# B&R Automation Studio project A2019059_Linka_Power_CP (part 18)

```iecst
            P1_Robot.KOM_OUT.ManipSrobovania_BezpecnaPozicia:= FALSE;

            P1_Srobovanie.PAR.OsX_ZadanaPozicia:= P1_RemPremenne.P1_Srob5F_PozX_ZadnejSkrutkyM4; //mm
            P1_Srobovanie.PAR.OsY_ZadanaPozicia:= P1_RemPremenne.P1_Srob5F_PozY_ZadnejSkrutkyM4; //mm

            IF NOT SC_P1_Srobovanie.Switch1 AND SC_OvlManipulatora_OsX.Step = 1 AND P1_Srobovacky_VychodziaPozicia AND Safety.STAV.P1_ZonaBunky_AKTIVNA THEN
                OsX_POLOHUJ:= TRUE;
                SC_P1_Srobovanie.Switch1:= TRUE;
            END_IF

            IF NOT SC_P1_Srobovanie.Switch2 AND SC_OvlManipulatora_OsY.Step = 1 AND P1_Srobovacky_VychodziaPozicia AND (P1_Srobovanie.ServoManipulOsX_M20.STATUS.ActualPosition > 14) AND Safety.STAV.P1_ZonaBunky_AKTIVNA THEN
                OsY_POLOHUJ:= TRUE;
                SC_P1_Srobovanie.Switch2:= TRUE;
            END_IF

            IF P1_Srobovanie.STAV.OsX_PoziciaDosiahnuta AND P1_Srobovanie.STAV.OsY_PoziciaDosiahnuta THEN
                P1_Srobovanie.STAV.OsX_PoziciaDosiahnuta:= FALSE;
                P1_Srobovanie.STAV.OsY_PoziciaDosiahnuta:= FALSE;
                IF P1_Srobovanie.RR_PolohujNaPoziciuSkrutky_5F THEN
                    P1_Srobovanie.RR_PolohujNaPoziciuSkrutky_5F:= FALSE;
                    P1_Srobovanie.RR_PolohujNaPoziciuSkrutky_4F:= FALSE;
                    P1_Srobovanie.RR_PolohujNaPoziciuSkrutky_5H:= FALSE;
                    SC_P1_Srobovanie.ResetStep:= TRUE;
                    SC_P1_Srobovanie.Step:= 700;
                ELSE
                    SC_P1_Srobovanie.ResetStep:= TRUE;
                    SC_P1_Srobovanie.Step:= 243;
                END_IF
            END_IF

        243:
            SC_P1_Srobovanie.StepName:='243 - Automaticky Rezim - model 5F, vymazanie vysledkov srobovania';
            SC_P1_Srobovanie.IdleTime.PT:= T#2s;
            SC_P1_Srobovanie.AlarmTime.PT:= T#5s;

            IF NOT SC_P1_Srobovanie.Switch1 THEN
                P1_Srobovanie.Skrutkovacka_M4.RESET_Vysledkov:= TRUE;
                SC_P1_Srobovanie.Switch1:= TRUE;
            END_IF

            IF NOT P1_Srobovanie.Skrutkovacka_M4.Stav_VysledokUtahovania_NG AND NOT P1_Srobovanie.Skrutkovacka_M4.Stav_VysledokUtahovania_OK AND NOT P1_Srobovanie.Skrutkovacka_M4.Stav_UtahovanieUkoncene THEN
                P1_Srobovanie.Skrutkovacka_M4.RESET_Vysledkov:= FALSE;
                SC_P1_Srobovanie.ResetStep:= TRUE;
                SC_P1_Srobovanie.Step:= 245;
            END_IF

        245:
            SC_P1_Srobovanie.StepName:='245 - Automaticky Rezim - model 5F, kontrola skrutky M4 v skrutkovacke';
            SC_P1_Srobovanie.IdleTime.PT:= T#5s;
            SC_P1_Srobovanie.AlarmTime.PT:= T#10s;
            SC_P1_Srobovanie.AlarmTime.IN:= TRUE;

            IF P1_Srobovanie.SkrutkovaciSet_M4.SkrutkaM4_Pripravena AND P1_Srobovanie.Skrutkovacka_M4.Stav_READY_to_START THEN
                SC_P1_Srobovanie.ResetStep:= TRUE;
                SC_P1_Srobovanie.Step:= 248;
            ELSIF SC_P1_Srobovanie.AlarmTime.Q THEN
                IF NOT P1_Srobovanie.Skrutkovacka_M4.Stav_READY_to_START THEN
                    P1_Alarmy[151]:= TRUE;
                    P1_StoperSrobovania.STAV.Porucha:= TRUE;
                    P1_Srobovanie.OUT.KOM_Srobovanie_Ukoncene:= TRUE;
                    SC_P1_Srobovanie.ResetStep:= TRUE;
                    SC_P1_Srobovanie.Step:= 258;
                ELSE
                    FazaNavratu:= 240;
                    SC_P1_Srobovanie.ResetStep:= TRUE;
                    SC_P1_Srobovanie.Step:= 510;
                END_IF
            END_IF

        248:
            SC_P1_Srobovanie.StepName:='248 - Automaticky Rezim - model 5F, vysunutie skrutkovacky M4';
            SC_P1_Srobovanie.IdleTime.PT:= T#500ms;
            SC_P1_Srobovanie.AlarmTime.PT:= T#10s;
            SC_P1_Srobovanie.IdleTime.IN:= TRUE;

            P1_Srobovanie.OUT.SkrutkM4_PrisavSkrutky_RUN_YV81:= TRUE;
            SC_P1_Srobovanie.AlarmTime.IN:= (P1_Srobovanie.IN.SkrutkM4_VysunutieHrotu_IOS10 < 1);

            IF NOT SC_P1_Srobovanie.Switch1 AND SC_P1_Srobovanie.IdleTime.Q THEN
                P1_Srobovanie.OUT.SkrutkM4_VYSUN_YV79:= TRUE;
                P1_Srobovanie.Skrutkovacka_M4.START_Utahovania:= TRUE;
                SC_P1_Srobovanie.Switch1:= TRUE;
            END_IF

            IF NOT P1_Srobovanie.Skrutkovacka_M4.Stav_UtahovanieUkoncene AND P1_Srobovanie.IN.SkrutkM4_VysunutieHrotu_IOS10 > 1 THEN
                SC_P1_Srobovanie.ResetStep:= TRUE;
                SC_P1_Srobovanie.Step:= 250;
            ELSIF SC_P1_Srobovanie.AlarmTime.Q THEN
                P1_Alarmy[144]:= TRUE;
                P1_Srobovanie.OUT.SkrutkM4_VYSUN_YV79:= FALSE;
                P1_Srobovanie.Skrutkovacka_M4.START_Utahovania:= FALSE;
                P1_StoperSrobovania.STAV.Porucha:= TRUE;
                P1_Srobovanie.OUT.KOM_Srobovanie_Ukoncene:= TRUE;
                SC_P1_Srobovanie.ResetStep:= TRUE;
                SC_P1_Srobovanie.Step:= 258;
            END_IF

        250:
            SC_P1_Srobovanie.StepName:='250 - Automaticky Rezim - model 5F, cakam na ukoncenie skrutkovania skrutkovacky M4';
            SC_P1_Srobovanie.IdleTime.PT:= T#30s;
            SC_P1_Srobovanie.AlarmTime.PT:= T#10s;
            SC_P1_Srobovanie.IdleTime.IN:= TRUE;
            SC_P1_Srobovanie.AlarmTime.IN:= TRUE;

            IF P1_Srobovanie.Skrutkovacka_M4.Stav_UtahovanieUkoncene THEN
                P1_Srobovanie.Skrutkovacka_M4.START_Utahovania:= FALSE;
                CasSrobovania:= TIME_TO_REAL(SC_P1_Srobovanie.IdleTime.ET);
                Reports.Skrutkovacky.VyskaSkrutkovania.P1_ZadnaSkrutkaM4:= REAL_TO_STRING(P1_Srobovanie.IN.SkrutkM4_VysunutieHrotu_IOS10);
                Reports.Skrutkovacky.CasSkrutkovania.P1_ZadnaSkrutkaM4:= REAL_TO_STRING(CasSrobovania/1000);
                SC_P1_Srobovanie.ResetStep:= TRUE;
                SC_P1_Srobovanie.Step:= 253;
            ELSIF SC_P1_Srobovanie.AlarmTime.Q THEN
                P1_Alarmy[148]:= TRUE;
                P1_Srobovanie.OUT.SkrutkM4_VYSUN_YV79:= FALSE;
                P1_Srobovanie.Skrutkovacka_M4.START_Utahovania:= FALSE;
                P1_StoperSrobovania.STAV.Porucha:= TRUE;
                P1_Srobovanie.OUT.KOM_Srobovanie_Ukoncene:= TRUE;
                SC_P1_Srobovanie.ResetStep:= TRUE;
                SC_P1_Srobovanie.Step:= 258;
            END_IF

        253:
            SC_P1_Srobovanie.StepName:='253 - Automaticky Rezim - model 5F, zasunutie skrutkovacky M4 a vypnutie prisavania skrutky';
            SC_P1_Srobovanie.IdleTime.PT:= T#200ms;
            SC_P1_Srobovanie.AlarmTime.PT:= T#5s;

            IF NOT SC_P1_Srobovanie.Switch1 THEN
                P1_Srobovanie.OUT.SkrutkM4_VYSUN_YV79:= FALSE;
                P1_Srobovanie.OUT.SkrutkM4_PrisavSkrutky_RUN_YV81:= FALSE;
                SC_P1_Srobovanie.Switch1:= TRUE;
            END_IF

            IF P1_Srobovanie.IN.SkrutkM4_ZASUNUTY_MS17 THEN
                SC_P1_Srobovanie.ResetStep:= TRUE;
                SC_P1_Srobovanie.Step:= 254;
            END_IF

        254:
            SC_P1_Srobovanie.StepName:='254 - Automaticky Rezim - model 5F, signal skrutka M4 odobrata';
            SC_P1_Srobovanie.IdleTime.PT:= T#200ms;
            SC_P1_Srobovanie.AlarmTime.PT:= T#5s;

            IF NOT SC_P1_Srobovanie.Switch1 THEN
                P1_Srobovanie.SkrutkovaciSet_M4.SkrutkaM4_Odobrata:= TRUE;
                SC_P1_Srobovanie.Switch1:= TRUE;
            END_IF

            IF NOT P1_Srobovanie.SkrutkovaciSet_M4.SkrutkaM4_Pripravena THEN
                P1_Srobovanie.SkrutkovaciSet_M4.SkrutkaM4_Odobrata:= FALSE;
                SC_P1_Srobovanie.ResetStep:= TRUE;
                SC_P1_Srobovanie.Step:= 255;
            END_IF

        255:
            SC_P1_Srobovanie.StepName:='255 - Automaticky Rezim - model 5F, kontrola vysledkov skrutkovania zadnej skrutky M4';
            SC_P1_Srobovanie.IdleTime.PT:= T#200ms;
            SC_P1_Srobovanie.AlarmTime.PT:= T#5s;

            IF P1_Srobovanie.Skrutkovacka_M4.Stav_VysledokUtahovania_OK THEN
                P1_Srobovanie.STAV.Vysledok_Srobovania:= 'OK';
                P1_Srobovanie.OUT.KOM_Srobovanie_Ukoncene:= TRUE;
                SC_P1_Srobovanie.ResetStep:= TRUE;
                SC_P1_Srobovanie.Step:= 258;
            ELSIF P1_Srobovanie.Skrutkovacka_M4.Stav_VysledokUtahovania_NG THEN
                P1_Srobovanie.STAV.Vysledok_Srobovania:= 'NG';
                P1_Srobovanie.OUT.KOM_Srobovanie_Ukoncene:= TRUE;
                SC_P1_Srobovanie.ResetStep:= TRUE;
                SC_P1_Srobovanie.Step:= 258;
            END_IF

        258:
            SC_P1_Srobovanie.StepName:='258 - Automaticky Rezim - model 5F, cakam na zrusenie signalu zaskrutkuj zadnu skrutku M4';
            SC_P1_Srobovanie.IdleTime.PT:= T#200ms;
            SC_P1_Srobovanie.AlarmTime.PT:= T#5s;

            IF NOT P1_StoperSrobovania.OUT.KOM_5F_ZasrobujZadnuSkrutku_M4 THEN
                P1_Srobovanie.OUT.KOM_Srobovanie_Ukoncene:= FALSE;
                SC_P1_Srobovanie.ResetStep:= TRUE;
                SC_P1_Srobovanie.Step:= 100;
            END_IF

            //Zaskrutkovanie prednej skrutky M4//

        260:
            SC_P1_Srobovanie.StepName:='260 - Automaticky Rezim - model 5F, napolohovanie zadnej skrutkovacky M4 na poziciu prednej skrutky M4';
            SC_P1_Srobovanie.IdleTime.PT:= T#200ms;
            SC_P1_Srobovanie.AlarmTime.PT:= T#5s;

            P1_Robot.KOM_OUT.ManipSrobovania_BezpecnaPozicia:= FALSE;

            P1_Srobovanie.PAR.OsX_ZadanaPozicia:= P1_RemPremenne.P1_Srob5F_PozX_PrednejSkrutkyM4; //mm
            P1_Srobovanie.PAR.OsY_ZadanaPozicia:= P1_RemPremenne.P1_Srob5F_PozY_PrednejSkrutkyM4; //mm

            IF NOT SC_P1_Srobovanie.Switch1 AND SC_OvlManipulatora_OsX.Step = 1 AND P1_Srobovacky_VychodziaPozicia AND Safety.STAV.P1_ZonaBunky_AKTIVNA THEN
                OsX_POLOHUJ:= TRUE;
                SC_P1_Srobovanie.Switch1:= TRUE;
            END_IF

            IF NOT SC_P1_Srobovanie.Switch2 AND SC_OvlManipulatora_OsY.Step = 1 AND P1_Srobovacky_VychodziaPozicia AND (P1_Srobovanie.ServoManipulOsX_M20.STATUS.ActualPosition > 14) AND Safety.STAV.P1_ZonaBunky_AKTIVNA THEN
                OsY_POLOHUJ:= TRUE;
                SC_P1_Srobovanie.Switch2:= TRUE;
            END_IF

            IF P1_Srobovanie.STAV.OsX_PoziciaDosiahnuta AND P1_Srobovanie.STAV.OsY_PoziciaDosiahnuta THEN
                P1_Srobovanie.STAV.OsX_PoziciaDosiahnuta:= FALSE;
                P1_Srobovanie.STAV.OsY_PoziciaDosiahnuta:= FALSE;
                IF P1_Srobovanie.RR_PolohujNaPoziciuSkrutky_5F THEN
                    P1_Srobovanie.RR_PolohujNaPoziciuSkrutky_5F:= FALSE;
                    P1_Srobovanie.RR_PolohujNaPoziciuSkrutky_4F:= FALSE;
                    P1_Srobovanie.RR_PolohujNaPoziciuSkrutky_5H:= FALSE;
                    SC_P1_Srobovanie.ResetStep:= TRUE;
                    SC_P1_Srobovanie.Step:= 700;
                ELSE
                    SC_P1_Srobovanie.ResetStep:= TRUE;
                    SC_P1_Srobovanie.Step:= 263;
                END_IF
            END_IF

        263:
            SC_P1_Srobovanie.StepName:='263 - Automaticky Rezim - model 5F, vymazanie vysledkov srobovania';
            SC_P1_Srobovanie.IdleTime.PT:= T#2s;
            SC_P1_Srobovanie.AlarmTime.PT:= T#5s;

            IF NOT SC_P1_Srobovanie.Switch1 THEN
                P1_Srobovanie.Skrutkovacka_M4.RESET_Vysledkov:= TRUE;
                SC_P1_Srobovanie.Switch1:= TRUE;
            END_IF

            IF NOT P1_Srobovanie.Skrutkovacka_M4.Stav_VysledokUtahovania_NG AND NOT P1_Srobovanie.Skrutkovacka_M4.Stav_VysledokUtahovania_OK AND NOT P1_Srobovanie.Skrutkovacka_M4.Stav_UtahovanieUkoncene THEN
                P1_Srobovanie.Skrutkovacka_M4.RESET_Vysledkov:= FALSE;
                SC_P1_Srobovanie.ResetStep:= TRUE;
                SC_P1_Srobovanie.Step:= 265;
            END_IF

        265:
            SC_P1_Srobovanie.StepName:='265 - Automaticky Rezim - model 5F, kontrola skrutky M4 v skrutkovacke';
            SC_P1_Srobovanie.IdleTime.PT:= T#5s;
            SC_P1_Srobovanie.AlarmTime.PT:= T#10s;
            SC_P1_Srobovanie.AlarmTime.IN:= TRUE;

            IF P1_Srobovanie.SkrutkovaciSet_M4.SkrutkaM4_Pripravena AND P1_Srobovanie.Skrutkovacka_M4.Stav_READY_to_START THEN
                SC_P1_Srobovanie.ResetStep:= TRUE;
                SC_P1_Srobovanie.Step:= 268;
            ELSIF SC_P1_Srobovanie.AlarmTime.Q THEN
                IF NOT P1_Srobovanie.Skrutkovacka_M4.Stav_READY_to_START THEN
                    P1_Alarmy[151]:= TRUE;
                    P1_StoperSrobovania.STAV.Porucha:= TRUE;
                    P1_Srobovanie.OUT.KOM_Srobovanie_Ukoncene:= TRUE;
                    SC_P1_Srobovanie.ResetStep:= TRUE;
                    SC_P1_Srobovanie.Step:= 278;
                ELSE
                    FazaNavratu:= 260;
                    SC_P1_Srobovanie.ResetStep:= TRUE;
                    SC_P1_Srobovanie.Step:= 510;
                END_IF
            END_IF

        268:
            SC_P1_Srobovanie.StepName:='268 - Automaticky Rezim - model 5F, vysunutie skrutkovacky M4';
            SC_P1_Srobovanie.IdleTime.PT:= T#500ms;
            SC_P1_Srobovanie.AlarmTime.PT:= T#10s;
            SC_P1_Srobovanie.IdleTime.IN:= TRUE;

            P1_Srobovanie.OUT.SkrutkM4_PrisavSkrutky_RUN_YV81:= TRUE;
            SC_P1_Srobovanie.AlarmTime.IN:= (P1_Srobovanie.IN.SkrutkM4_VysunutieHrotu_IOS10 < 1);

            IF NOT SC_P1_Srobovanie.Switch1 AND SC_P1_Srobovanie.IdleTime.Q THEN
                P1_Srobovanie.OUT.SkrutkM4_VYSUN_YV79:= TRUE;
                P1_Srobovanie.Skrutkovacka_M4.START_Utahovania:= TRUE;
                SC_P1_Srobovanie.Switch1:= TRUE;
            END_IF

            IF NOT P1_Srobovanie.Skrutkovacka_M4.Stav_UtahovanieUkoncene AND P1_Srobovanie.IN.SkrutkM4_VysunutieHrotu_IOS10 > 1 THEN
                SC_P1_Srobovanie.ResetStep:= TRUE;
                SC_P1_Srobovanie.Step:= 270;
            ELSIF SC_P1_Srobovanie.AlarmTime.Q THEN
                P1_Alarmy[144]:= TRUE;
                P1_Srobovanie.OUT.SkrutkM4_VYSUN_YV79:= FALSE;
                P1_Srobovanie.Skrutkovacka_M4.START_Utahovania:= FALSE;
                P1_StoperSrobovania.STAV.Porucha:= TRUE;
                P1_Srobovanie.OUT.KOM_Srobovanie_Ukoncene:= TRUE;
                SC_P1_Srobovanie.ResetStep:= TRUE;
                SC_P1_Srobovanie.Step:= 278;
            END_IF

        270:
            SC_P1_Srobovanie.StepName:='270 - Automaticky Rezim - model 5F, cakam na ukoncenie skrutkovania skrutkovacky M4';
            SC_P1_Srobovanie.IdleTime.PT:= T#30s;
            SC_P1_Srobovanie.AlarmTime.PT:= T#10s;
            SC_P1_Srobovanie.IdleTime.IN:= TRUE;
            SC_P1_Srobovanie.AlarmTime.IN:= TRUE;

            IF P1_Srobovanie.Skrutkovacka_M4.Stav_UtahovanieUkoncene THEN
                P1_Srobovanie.Skrutkovacka_M4.START_Utahovania:= FALSE;
                CasSrobovania:= TIME_TO_REAL(SC_P1_Srobovanie.IdleTime.ET);
                Reports.Skrutkovacky.VyskaSkrutkovania.P1_PrednaSkrutkaM4:= REAL_TO_STRING(P1_Srobovanie.IN.SkrutkM4_VysunutieHrotu_IOS10);
                Reports.Skrutkovacky.CasSkrutkovania.P1_PrednaSkrutkaM4:= REAL_TO_STRING(CasSrobovania/1000);
                SC_P1_Srobovanie.ResetStep:= TRUE;
                SC_P1_Srobovanie.Step:= 273;
            ELSIF SC_P1_Srobovanie.AlarmTime.Q THEN
                P1_Alarmy[148]:= TRUE;
                P1_Srobovanie.OUT.SkrutkM4_VYSUN_YV79:= FALSE;
                P1_Srobovanie.Skrutkovacka_M4.START_Utahovania:= FALSE;
                P1_StoperSrobovania.STAV.Porucha:= TRUE;
                P1_Srobovanie.OUT.KOM_Srobovanie_Ukoncene:= TRUE;
                SC_P1_Srobovanie.ResetStep:= TRUE;
                SC_P1_Srobovanie.Step:= 278;
            END_IF

        273:
            SC_P1_Srobovanie.StepName:='273 - Automaticky Rezim - model 5F, zasunutie skrutkovacky M4 a vypnutie prisavania skrutky';
            SC_P1_Srobovanie.IdleTime.PT:= T#200ms;
            SC_P1_Srobovanie.AlarmTime.PT:= T#5s;

            IF NOT SC_P1_Srobovanie.Switch1 THEN
                P1_Srobovanie.OUT.SkrutkM4_VYSUN_YV79:= FALSE;
                P1_Srobovanie.OUT.SkrutkM4_PrisavSkrutky_RUN_YV81:= FALSE;
                SC_P1_Srobovanie.Switch1:= TRUE;
            END_IF

            IF P1_Srobovanie.IN.SkrutkM4_ZASUNUTY_MS17 THEN
                SC_P1_Srobovanie.ResetStep:= TRUE;
                SC_P1_Srobovanie.Step:= 274;
            END_IF

        274:
            SC_P1_Srobovanie.StepName:='274 - Automaticky Rezim - model 5F, signal skrutka M4 odobrata';
            SC_P1_Srobovanie.IdleTime.PT:= T#200ms;
            SC_P1_Srobovanie.AlarmTime.PT:= T#5s;

            IF NOT SC_P1_Srobovanie.Switch1 THEN
                P1_Srobovanie.SkrutkovaciSet_M4.SkrutkaM4_Odobrata:= TRUE;
                SC_P1_Srobovanie.Switch1:= TRUE;
            END_IF

            IF NOT P1_Srobovanie.SkrutkovaciSet_M4.SkrutkaM4_Pripravena THEN
                P1_Srobovanie.SkrutkovaciSet_M4.SkrutkaM4_Odobrata:= FALSE;
                SC_P1_Srobovanie.ResetStep:= TRUE;
                SC_P1_Srobovanie.Step:= 275;
            END_IF

        275:
            SC_P1_Srobovanie.StepName:='275 - Automaticky Rezim - model 5F, kontrola vysledkov skrutkovania prednej skrutky M4';
            SC_P1_Srobovanie.IdleTime.PT:= T#200ms;
            SC_P1_Srobovanie.AlarmTime.PT:= T#5s;

            IF P1_Srobovanie.Skrutkovacka_M4.Stav_VysledokUtahovania_OK THEN
                P1_Srobovanie.STAV.Vysledok_Srobovania:= 'OK';
                P1_Srobovanie.OUT.KOM_Srobovanie_Ukoncene:= TRUE;
                SC_P1_Srobovanie.ResetStep:= TRUE;
                SC_P1_Srobovanie.Step:= 278;
            ELSIF P1_Srobovanie.Skrutkovacka_M4.Stav_VysledokUtahovania_NG THEN
                P1_Srobovanie.STAV.Vysledok_Srobovania:= 'NG';
                P1_Srobovanie.OUT.KOM_Srobovanie_Ukoncene:= TRUE;
                SC_P1_Srobovanie.ResetStep:= TRUE;
                SC_P1_Srobovanie.Step:= 278;
            END_IF

        278:
            SC_P1_Srobovanie.StepName:='278 - Automaticky Rezim - model 5F, cakam na zrusenie signalu zaskrutkuj prednu skrutku M4';
            SC_P1_Srobovanie.IdleTime.PT:= T#200ms;
            SC_P1_Srobovanie.AlarmTime.PT:= T#5s;

            IF NOT P1_StoperSrobovania.OUT.KOM_5F_ZasrobujPrednuSkrutku_M4 THEN
                P1_Srobovanie.OUT.KOM_Srobovanie_Ukoncene:= FALSE;
                SC_P1_Srobovanie.ResetStep:= TRUE;
                SC_P1_Srobovanie.Step:= 100;
            END_IF

            //Zaskrutkovanie skrutky M4 pre DPS//

        280:
            SC_P1_Srobovanie.StepName:='280 - Automaticky Rezim - model 5F, napolohovanie zadnej skrutkovacky M4 na poziciu  skrutky M4 pre DPS';
            SC_P1_Srobovanie.IdleTime.PT:= T#200ms;
            SC_P1_Srobovanie.AlarmTime.PT:= T#5s;

            P1_Robot.KOM_OUT.ManipSrobovania_BezpecnaPozicia:= FALSE;

            P1_Srobovanie.PAR.OsX_ZadanaPozicia:= P1_RemPremenne.P1_Srob5F_PozX_SkrutkyDPS_M4; //mm
            P1_Srobovanie.PAR.OsY_ZadanaPozicia:= P1_RemPremenne.P1_Srob5F_PozY_SkrutkyDPS_M4; //mm

            IF NOT SC_P1_Srobovanie.Switch1 AND SC_OvlManipulatora_OsX.Step = 1 AND P1_Srobovacky_VychodziaPozicia AND Safety.STAV.P1_ZonaBunky_AKTIVNA THEN
                OsX_POLOHUJ:= TRUE;
                SC_P1_Srobovanie.Switch1:= TRUE;
            END_IF

            IF NOT SC_P1_Srobovanie.Switch2 AND SC_OvlManipulatora_OsY.Step = 1 AND P1_Srobovacky_VychodziaPozicia AND (P1_Srobovanie.ServoManipulOsX_M20.STATUS.ActualPosition > 14) AND Safety.STAV.P1_ZonaBunky_AKTIVNA THEN
                OsY_POLOHUJ:= TRUE;
                SC_P1_Srobovanie.Switch2:= TRUE;
            END_IF

            IF P1_Srobovanie.STAV.OsX_PoziciaDosiahnuta AND P1_Srobovanie.STAV.OsY_PoziciaDosiahnuta THEN
                P1_Srobovanie.STAV.OsX_PoziciaDosiahnuta:= FALSE;
                P1_Srobovanie.STAV.OsY_PoziciaDosiahnuta:= FALSE;
                IF P1_Srobovanie.RR_PolohujNaPoziciuSkrutky_5F THEN
                    P1_Srobovanie.RR_PolohujNaPoziciuSkrutky_5F:= FALSE;
                    P1_Srobovanie.RR_PolohujNaPoziciuSkrutky_4F:= FALSE;
                    P1_Srobovanie.RR_PolohujNaPoziciuSkrutky_5H:= FALSE;
                    SC_P1_Srobovanie.ResetStep:= TRUE;
                    SC_P1_Srobovanie.Step:= 700;
                ELSE
                    SC_P1_Srobovanie.ResetStep:= TRUE;
                    SC_P1_Srobovanie.Step:= 282;
                END_IF
            END_IF

        282:
            SC_P1_Srobovanie.StepName:='282 - Automaticky Rezim - model 5F, vymazanie vysledkov srobovania';
            SC_P1_Srobovanie.IdleTime.PT:= T#2s;
            SC_P1_Srobovanie.AlarmTime.PT:= T#5s;

            IF NOT SC_P1_Srobovanie.Switch1 THEN
                P1_Srobovanie.Skrutkovacka_M4.RESET_Vysledkov:= TRUE;
                SC_P1_Srobovanie.Switch1:= TRUE;
            END_IF

            IF NOT P1_Srobovanie.Skrutkovacka_M4.Stav_VysledokUtahovania_NG AND NOT P1_Srobovanie.Skrutkovacka_M4.Stav_VysledokUtahovania_OK AND NOT P1_Srobovanie.Skrutkovacka_M4.Stav_UtahovanieUkoncene THEN
                P1_Srobovanie.Skrutkovacka_M4.RESET_Vysledkov:= FALSE;
                SC_P1_Srobovanie.ResetStep:= TRUE;
                SC_P1_Srobovanie.Step:= 283;
            END_IF

        283:
            SC_P1_Srobovanie.StepName:='283 - Automaticky Rezim - model 5F, kontrola skrutky M4 v skrutkovacke';
            SC_P1_Srobovanie.IdleTime.PT:= T#5s;
            SC_P1_Srobovanie.AlarmTime.PT:= T#10s;
            SC_P1_Srobovanie.AlarmTime.IN:= TRUE;

            IF P1_Srobovanie.SkrutkovaciSet_M4.SkrutkaM4_Pripravena AND P1_Srobovanie.Skrutkovacka_M4.Stav_READY_to_START THEN
                SC_P1_Srobovanie.ResetStep:= TRUE;
                SC_P1_Srobovanie.Step:= 284;
            ELSIF SC_P1_Srobovanie.AlarmTime.Q THEN
                IF NOT P1_Srobovanie.Skrutkovacka_M4.Stav_READY_to_START THEN
                    P1_Alarmy[151]:= TRUE;
                    P1_StoperSrobovania.STAV.Porucha:= TRUE;
                    P1_Srobovanie.OUT.KOM_Srobovanie_Ukoncene:= TRUE;
                    SC_P1_Srobovanie.ResetStep:= TRUE;
                    SC_P1_Srobovanie.Step:= 289;
                ELSE
                    FazaNavratu:= 280;
                    SC_P1_Srobovanie.ResetStep:= TRUE;
                    SC_P1_Srobovanie.Step:= 510;
                END_IF
            END_IF

        284:
            SC_P1_Srobovanie.StepName:='284 - Automaticky Rezim - model 5F, vysunutie skrutkovacky M4';
            SC_P1_Srobovanie.IdleTime.PT:= T#500ms;
            SC_P1_Srobovanie.AlarmTime.PT:= T#10s;
            SC_P1_Srobovanie.IdleTime.IN:= TRUE;

            P1_Srobovanie.OUT.SkrutkM4_PrisavSkrutky_RUN_YV81:= TRUE;
            SC_P1_Srobovanie.AlarmTime.IN:= (P1_Srobovanie.IN.SkrutkM4_VysunutieHrotu_IOS10 < 1);

            IF NOT SC_P1_Srobovanie.Switch1 AND SC_P1_Srobovanie.IdleTime.Q THEN
                P1_Srobovanie.OUT.SkrutkM4_VYSUN_YV79:= TRUE;
                P1_Srobovanie.Skrutkovacka_M4.START_Utahovania:= TRUE;
                SC_P1_Srobovanie.Switch1:= TRUE;
            END_IF

            IF NOT P1_Srobovanie.Skrutkovacka_M4.Stav_UtahovanieUkoncene AND P1_Srobovanie.IN.SkrutkM4_VysunutieHrotu_IOS10 > 1 AND NOT TEST THEN
                SC_P1_Srobovanie.ResetStep:= TRUE;
                SC_P1_Srobovanie.Step:= 285;
            ELSIF SC_P1_Srobovanie.AlarmTime.Q AND NOT TEST THEN
                P1_Alarmy[144]:= TRUE;
                P1_Srobovanie.OUT.SkrutkM4_VYSUN_YV79:= FALSE;
                P1_Srobovanie.Skrutkovacka_M4.START_Utahovania:= FALSE;
                P1_StoperSrobovania.STAV.Porucha:= TRUE;
                P1_Srobovanie.OUT.KOM_Srobovanie_Ukoncene:= TRUE;
                SC_P1_Srobovanie.ResetStep:= TRUE;
                SC_P1_Srobovanie.Step:= 289;
            END_IF

        285:
            SC_P1_Srobovanie.StepName:='285 - Automaticky Rezim - model 5F, cakam na ukoncenie skrutkovania skrutkovacky M4';
            SC_P1_Srobovanie.IdleTime.PT:= T#30s;
            SC_P1_Srobovanie.AlarmTime.PT:= T#10s;
            SC_P1_Srobovanie.IdleTime.IN:= TRUE;
            SC_P1_Srobovanie.AlarmTime.IN:= TRUE;

            IF P1_Srobovanie.Skrutkovacka_M4.Stav_UtahovanieUkoncene THEN
                P1_Srobovanie.Skrutkovacka_M4.START_Utahovania:= FALSE;
                CasSrobovania:= TIME_TO_REAL(SC_P1_Srobovanie.IdleTime.ET);
                Reports.Skrutkovacky.VyskaSkrutkovania.P1_SkrutkaDPS_M4:= REAL_TO_STRING(P1_Srobovanie.IN.SkrutkM4_VysunutieHrotu_IOS10);
                Reports.Skrutkovacky.CasSkrutkovania.P1_SkrutkaDPS_M4:= REAL_TO_STRING(CasSrobovania/1000);
                SC_P1_Srobovanie.ResetStep:= TRUE;
                SC_P1_Srobovanie.Step:= 286;
            ELSIF SC_P1_Srobovanie.AlarmTime.Q THEN
                P1_Alarmy[148]:= TRUE;
                P1_Srobovanie.OUT.SkrutkM4_VYSUN_YV79:= FALSE;
                P1_Srobovanie.Skrutkovacka_M4.START_Utahovania:= FALSE;
                P1_StoperSrobovania.STAV.Porucha:= TRUE;
                P1_Srobovanie.OUT.KOM_Srobovanie_Ukoncene:= TRUE;
                SC_P1_Srobovanie.ResetStep:= TRUE;
                SC_P1_Srobovanie.Step:= 289;
            END_IF

        286:
            SC_P1_Srobovanie.StepName:='286 - Automaticky Rezim - model 5F, zasunutie skrutkovacky M4 a vypnutie prisavania skrutky';
            SC_P1_Srobovanie.IdleTime.PT:= T#200ms;
            SC_P1_Srobovanie.AlarmTime.PT:= T#5s;

            IF NOT SC_P1_Srobovanie.Switch1 THEN
                P1_Srobovanie.OUT.SkrutkM4_VYSUN_YV79:= FALSE;
                P1_Srobovanie.OUT.SkrutkM4_PrisavSkrutky_RUN_YV81:= FALSE;
                SC_P1_Srobovanie.Switch1:= TRUE;
            END_IF

            IF P1_Srobovanie.IN.SkrutkM4_ZASUNUTY_MS17 THEN
                SC_P1_Srobovanie.ResetStep:= TRUE;
                SC_P1_Srobovanie.Step:= 287;
            END_IF

        287:
            SC_P1_Srobovanie.StepName:='287 - Automaticky Rezim - model 5F, signal skrutka M4 odobrata';
            SC_P1_Srobovanie.IdleTime.PT:= T#200ms;
            SC_P1_Srobovanie.AlarmTime.PT:= T#5s;

            IF NOT SC_P1_Srobovanie.Switch1 THEN
                P1_Srobovanie.SkrutkovaciSet_M4.SkrutkaM4_Odobrata:= TRUE;
                SC_P1_Srobovanie.Switch1:= TRUE;
            END_IF

            IF NOT P1_Srobovanie.SkrutkovaciSet_M4.SkrutkaM4_Pripravena THEN
                P1_Srobovanie.SkrutkovaciSet_M4.SkrutkaM4_Odobrata:= FALSE;
                SC_P1_Srobovanie.ResetStep:= TRUE;
                SC_P1_Srobovanie.Step:= 288;
            END_IF

        288:
            SC_P1_Srobovanie.StepName:='288 - Automaticky Rezim - model 5F, kontrola vysledkov skrutkovania skrutky M4 pre DPS';
            SC_P1_Srobovanie.IdleTime.PT:= T#200ms;
            SC_P1_Srobovanie.AlarmTime.PT:= T#5s;

            IF P1_Srobovanie.Skrutkovacka_M4.Stav_VysledokUtahovania_OK THEN
                P1_Srobovanie.STAV.Vysledok_Srobovania:= 'OK';
                P1_Srobovanie.OUT.KOM_Srobovanie_Ukoncene:= TRUE;
                SC_P1_Srobovanie.ResetStep:= TRUE;
                SC_P1_Srobovanie.Step:= 289;
            ELSIF P1_Srobovanie.Skrutkovacka_M4.Stav_VysledokUtahovania_NG THEN
                P1_Srobovanie.STAV.Vysledok_Srobovania:= 'NG';
                P1_Srobovanie.OUT.KOM_Srobovanie_Ukoncene:= TRUE;
                SC_P1_Srobovanie.ResetStep:= TRUE;
                SC_P1_Srobovanie.Step:= 289;
            END_IF

        289:
            SC_P1_Srobovanie.StepName:='289 - Automaticky Rezim - model 5F, cakam na zrusenie signalu zaskrutkuj skrutku M4 pre DPS';
            SC_P1_Srobovanie.IdleTime.PT:= T#200ms;
            SC_P1_Srobovanie.AlarmTime.PT:= T#5s;

            IF NOT P1_StoperSrobovania.OUT.KOM_5F_ZasrobujSkrutkuDPS_M4 THEN
                P1_Srobovanie.OUT.KOM_Srobovanie_Ukoncene:= FALSE;
                SC_P1_Srobovanie.ResetStep:= TRUE;
                SC_P1_Srobovanie.Step:= 100;
            END_IF

            //**********************************************************************Model 5H*******************************************************************************************//
            //Zaskrutkovanie lavej skrutky K30//
        300:
            SC_P1_Srobovanie.StepName:='300 - Automaticky Rezim - model 5H, napolohovanie prednej skrutkovacky K30 na poziciu lavej skrutky K30';
            SC_P1_Srobovanie.IdleTime.PT:= T#200ms;
            SC_P1_Srobovanie.AlarmTime.PT:= T#5s;

            P1_Robot.KOM_OUT.ManipSrobovania_BezpecnaPozicia:= FALSE;

            P1_Srobovanie.PAR.OsX_ZadanaPozicia:= P1_RemPremenne.P1_Srob5H_PozX_LavejSkrutkyK30; //mm
            P1_Srobovanie.PAR.OsY_ZadanaPozicia:= P1_RemPremenne.P1_Srob5H_PozY_LavejSkrutkyK30; //mm

            IF NOT SC_P1_Srobovanie.Switch1 AND SC_OvlManipulatora_OsX.Step = 1 AND P1_Srobovacky_VychodziaPozicia AND Safety.STAV.P1_ZonaBunky_AKTIVNA THEN
                OsX_POLOHUJ:= TRUE;
                SC_P1_Srobovanie.Switch1:= TRUE;
            END_IF

            IF NOT SC_P1_Srobovanie.Switch2 AND SC_OvlManipulatora_OsY.Step = 1 AND P1_Srobovacky_VychodziaPozicia AND (P1_Srobovanie.ServoManipulOsX_M20.STATUS.ActualPosition > 14) AND Safety.STAV.P1_ZonaBunky_AKTIVNA THEN
                OsY_POLOHUJ:= TRUE;
                SC_P1_Srobovanie.Switch2:= TRUE;
            END_IF

            IF P1_Srobovanie.STAV.OsX_PoziciaDosiahnuta AND P1_Srobovanie.STAV.OsY_PoziciaDosiahnuta  THEN
                P1_Srobovanie.STAV.OsX_PoziciaDosiahnuta:= FALSE;
                P1_Srobovanie.STAV.OsY_PoziciaDosiahnuta:= FALSE;
                IF P1_Srobovanie.RR_PolohujNaPoziciuSkrutky_5H THEN
                    P1_Srobovanie.RR_PolohujNaPoziciuSkrutky_5H:= FALSE;
                    P1_Srobovanie.RR_PolohujNaPoziciuSkrutky_4F:= FALSE;
                    P1_Srobovanie.RR_PolohujNaPoziciuSkrutky_5F:= FALSE;
                    SC_P1_Srobovanie.ResetStep:= TRUE;
                    SC_P1_Srobovanie.Step:= 700;
                ELSE
                    SC_P1_Srobovanie.ResetStep:= TRUE;
                    SC_P1_Srobovanie.Step:= 303;
                END_IF
            END_IF

        303:
            SC_P1_Srobovanie.StepName:='303 - Automaticky Rezim - model 5H, vymazanie vysledkov srobovania';
            SC_P1_Srobovanie.IdleTime.PT:= T#2s;
            SC_P1_Srobovanie.AlarmTime.PT:= T#5s;

            IF NOT SC_P1_Srobovanie.Switch1 THEN
                P1_Srobovanie.Skrutkovacka_K30.RESET_Vysledkov:= TRUE;
                SC_P1_Srobovanie.Switch1:= TRUE;
            END_IF

            IF NOT P1_Srobovanie.Skrutkovacka_K30.Stav_VysledokUtahovania_NG AND NOT P1_Srobovanie.Skrutkovacka_K30.Stav_VysledokUtahovania_OK AND NOT P1_Srobovanie.Skrutkovacka_K30.Stav_UtahovanieUkoncene THEN
                P1_Srobovanie.Skrutkovacka_K30.RESET_Vysledkov:= FALSE;
                SC_P1_Srobovanie.ResetStep:= TRUE;
                SC_P1_Srobovanie.Step:= 305;
            END_IF

        305:
            SC_P1_Srobovanie.StepName:='305 - Automaticky Rezim - model 5H, kontrola skrutky K30 v skrutkovacke';
            SC_P1_Srobovanie.IdleTime.PT:= T#5s;
            SC_P1_Srobovanie.AlarmTime.PT:= T#10s;
            SC_P1_Srobovanie.AlarmTime.IN:= TRUE;

            IF P1_Srobovanie.SkrutkovaciSet_K30.SkrutkaK30_Pripravena AND P1_Srobovanie.Skrutkovacka_K30.Stav_READY_to_START THEN
                SC_P1_Srobovanie.ResetStep:= TRUE;
                SC_P1_Srobovanie.Step:= 308;
            ELSIF SC_P1_Srobovanie.AlarmTime.Q THEN
                IF NOT P1_Srobovanie.Skrutkovacka_K30.Stav_READY_to_START THEN
                    P1_Alarmy[149]:= TRUE;
                    P1_StoperSrobovania.STAV.Porucha:= TRUE;
                    P1_Srobovanie.OUT.KOM_Srobovanie_Ukoncene:= TRUE;
                    SC_P1_Srobovanie.ResetStep:= TRUE;
                    SC_P1_Srobovanie.Step:= 318;
                ELSE
                    FazaNavratu:= 300;
                    SC_P1_Srobovanie.ResetStep:= TRUE;
                    SC_P1_Srobovanie.Step:= 500;
                END_IF
            END_IF

        308:
            SC_P1_Srobovanie.StepName:='308 - Automaticky Rezim - model 5H, vysunutie skrutkovacky K30';
            SC_P1_Srobovanie.IdleTime.PT:= T#2s;
            SC_P1_Srobovanie.AlarmTime.PT:= T#5s;

            SC_P1_Srobovanie.AlarmTime.IN:= (P1_Srobovanie.IN.SkrutkK30_VysunutieHrotu_IOS8 < 2);

            IF NOT SC_P1_Srobovanie.Switch1 THEN
                P1_Srobovanie.OUT.SkrutkK30_PrisavSkrutky_RUN_YV90:= TRUE;
                P1_Srobovanie.Skrutkovacka_K30.START_Utahovania:= TRUE;
                P1_Srobovanie.OUT.SkrutkK30_VYSUN_YV89:= TRUE;
                SC_P1_Srobovanie.Switch1:= TRUE;
            ELSIF SC_P1_Srobovanie.AlarmTime.Q THEN
                P1_Alarmy[142]:= TRUE;
                P1_Srobovanie.OUT.SkrutkK30_VYSUN_YV89:= FALSE;
                P1_Srobovanie.Skrutkovacka_K30.START_Utahovania:= FALSE;
                P1_StoperSrobovania.STAV.Porucha:= TRUE;
                P1_Srobovanie.OUT.KOM_Srobovanie_Ukoncene:= TRUE;
                SC_P1_Srobovanie.ResetStep:= TRUE;
                SC_P1_Srobovanie.Step:= 318;
            END_IF

            IF NOT P1_Srobovanie.Skrutkovacka_K30.Stav_UtahovanieUkoncene AND P1_Srobovanie.IN.SkrutkK30_VysunutieHrotu_IOS8 > 2 THEN
                SC_P1_Srobovanie.ResetStep:= TRUE;
                SC_P1_Srobovanie.Step:= 310;
            END_IF

        310:
            SC_P1_Srobovanie.StepName:='310 - Automaticky Rezim - model 5H, cakam na ukoncenie skrutkovania skrutkovacky K30';
            SC_P1_Srobovanie.IdleTime.PT:= T#30s;
            SC_P1_Srobovanie.AlarmTime.PT:= T#10s;
            SC_P1_Srobovanie.IdleTime.IN:= TRUE;
            SC_P1_Srobovanie.AlarmTime.IN:= TRUE;

            IF P1_Srobovanie.Skrutkovacka_K30.Stav_UtahovanieUkoncene THEN
                P1_Srobovanie.Skrutkovacka_K30.START_Utahovania:= FALSE;
                CasSrobovania:= TIME_TO_REAL(SC_P1_Srobovanie.IdleTime.ET);
                Reports.Skrutkovacky.VyskaSkrutkovania.P1_LavaSkrutkaK30:= REAL_TO_STRING(P1_Srobovanie.IN.SkrutkK30_VysunutieHrotu_IOS8);
                Reports.Skrutkovacky.CasSkrutkovania.P1_LavaSkrutkaK30:= REAL_TO_STRING(CasSrobovania/1000);
                SC_P1_Srobovanie.ResetStep:= TRUE;
                SC_P1_Srobovanie.Step:= 313;
            ELSIF SC_P1_Srobovanie.AlarmTime.Q THEN
                P1_Alarmy[146]:= TRUE;
                P1_Srobovanie.OUT.SkrutkK30_VYSUN_YV89:= FALSE;
                P1_Srobovanie.Skrutkovacka_K30.START_Utahovania:= FALSE;
                P1_StoperSrobovania.STAV.Porucha:= TRUE;
                P1_Srobovanie.OUT.KOM_Srobovanie_Ukoncene:= TRUE;
                SC_P1_Srobovanie.ResetStep:= TRUE;
                SC_P1_Srobovanie.Step:= 318;
            END_IF

        313:
            SC_P1_Srobovanie.StepName:='313 - Automaticky Rezim - model 5H, zasunutie skrutkovacky K30 a vypnutie prisavania skrutky';
            SC_P1_Srobovanie.IdleTime.PT:= T#200ms;
            SC_P1_Srobovanie.AlarmTime.PT:= T#5s;

            IF NOT SC_P1_Srobovanie.Switch1 THEN
                P1_Srobovanie.OUT.SkrutkK30_VYSUN_YV89:= FALSE;
                P1_Srobovanie.OUT.SkrutkK30_PrisavSkrutky_RUN_YV90:= FALSE;
                SC_P1_Srobovanie.Switch1:= TRUE;
            END_IF

            IF P1_Srobovanie.IN.SkrutkK30_ZASUNUTY_MS20 THEN
                SC_P1_Srobovanie.ResetStep:= TRUE;
                SC_P1_Srobovanie.Step:= 314;
            END_IF

        314:
            SC_P1_Srobovanie.StepName:='314 - Automaticky Rezim - model 5H, signal skrutka K30 odobrata';
            SC_P1_Srobovanie.IdleTime.PT:= T#200ms;
            SC_P1_Srobovanie.AlarmTime.PT:= T#5s;

            IF NOT SC_P1_Srobovanie.Switch1 THEN
                P1_Srobovanie.SkrutkovaciSet_K30.SkrutkaK30_Odobrata:= TRUE;
                SC_P1_Srobovanie.Switch1:= TRUE;
            END_IF

            IF NOT P1_Srobovanie.SkrutkovaciSet_K30.SkrutkaK30_Pripravena THEN
                P1_Srobovanie.SkrutkovaciSet_K30.SkrutkaK30_Odobrata:= FALSE;
                SC_P1_Srobovanie.ResetStep:= TRUE;
                SC_P1_Srobovanie.Step:= 315;
            END_IF

        315:
            SC_P1_Srobovanie.StepName:='315 - Automaticky Rezim - model 5H, kontrola vysledkov skrutkovania lavej skrutky K30';
            SC_P1_Srobovanie.IdleTime.PT:= T#200ms;
            SC_P1_Srobovanie.AlarmTime.PT:= T#5s;

            IF P1_Srobovanie.Skrutkovacka_K30.Stav_VysledokUtahovania_OK THEN
                P1_Srobovanie.STAV.Vysledok_Srobovania:= 'OK';
                P1_Srobovanie.OUT.KOM_Srobovanie_Ukoncene:= TRUE;
                SC_P1_Srobovanie.ResetStep:= TRUE;
                SC_P1_Srobovanie.Step:= 318;
            ELSIF P1_Srobovanie.Skrutkovacka_K30.Stav_VysledokUtahovania_NG THEN
                P1_Srobovanie.STAV.Vysledok_Srobovania:= 'NG';
                P1_Srobovanie.OUT.KOM_Srobovanie_Ukoncene:= TRUE;
                SC_P1_Srobovanie.ResetStep:= TRUE;
                SC_P1_Srobovanie.Step:= 318;
            END_IF

        318:
            SC_P1_Srobovanie.StepName:='318 - Automaticky Rezim - model 5H, cakam na zrusenie signalu zaskrutkuj lavu skrutku K30';
            SC_P1_Srobovanie.IdleTime.PT:= T#200ms;
            SC_P1_Srobovanie.AlarmTime.PT:= T#5s;

            IF NOT P1_StoperSrobovania.OUT.KOM_5H_ZasrobujLavuSkrutku_K30 THEN
                P1_Srobovanie.OUT.KOM_Srobovanie_Ukoncene:= FALSE;
                SC_P1_Srobovanie.ResetStep:= TRUE;
                SC_P1_Srobovanie.Step:= 100;
            END_IF

            //Zaskrutkovanie pravej skrutky K30//

        320:
            SC_P1_Srobovanie.StepName:='320 - Automaticky Rezim - model 5H, napolohovanie prednej skrutkovacky K30 na poziciu pravej skrutky K30';
            SC_P1_Srobovanie.IdleTime.PT:= T#200ms;
            SC_P1_Srobovanie.AlarmTime.PT:= T#5s;

            P1_Robot.KOM_OUT.ManipSrobovania_BezpecnaPozicia:= FALSE;

            P1_Srobovanie.PAR.OsX_ZadanaPozicia:= P1_RemPremenne.P1_Srob5F_PozX_PravejSkrutkyK30; //mm
            P1_Srobovanie.PAR.OsY_ZadanaPozicia:= P1_RemPremenne.P1_Srob5F_PozY_PravejSkrutkyK30; //mm

            IF NOT SC_P1_Srobovanie.Switch1 AND SC_OvlManipulatora_OsX.Step = 1 AND P1_Srobovacky_VychodziaPozicia AND Safety.STAV.P1_ZonaBunky_AKTIVNA THEN
                OsX_POLOHUJ:= TRUE;
                SC_P1_Srobovanie.Switch1:= TRUE;
            END_IF

            IF NOT SC_P1_Srobovanie.Switch2 AND SC_OvlManipulatora_OsY.Step = 1 AND P1_Srobovacky_VychodziaPozicia AND (P1_Srobovanie.ServoManipulOsX_M20.STATUS.ActualPosition > 14) AND Safety.STAV.P1_ZonaBunky_AKTIVNA THEN
                OsY_POLOHUJ:= TRUE;
                SC_P1_Srobovanie.Switch2:= TRUE;
            END_IF

            IF P1_Srobovanie.STAV.OsX_PoziciaDosiahnuta AND P1_Srobovanie.STAV.OsY_PoziciaDosiahnuta  THEN
                P1_Srobovanie.STAV.OsX_PoziciaDosiahnuta:= FALSE;
                P1_Srobovanie.STAV.OsY_PoziciaDosiahnuta:= FALSE;
                IF P1_Srobovanie.RR_PolohujNaPoziciuSkrutky_5H THEN
                    P1_Srobovanie.RR_PolohujNaPoziciuSkrutky_5H:= FALSE;
                    P1_Srobovanie.RR_PolohujNaPoziciuSkrutky_4F:= FALSE;
                    P1_Srobovanie.RR_PolohujNaPoziciuSkrutky_5F:= FALSE;
                    SC_P1_Srobovanie.ResetStep:= TRUE;
                    SC_P1_Srobovanie.Step:= 700;
                ELSE
                    SC_P1_Srobovanie.ResetStep:= TRUE;
                    SC_P1_Srobovanie.Step:= 323;
                END_IF
            END_IF

        323:
            SC_P1_Srobovanie.StepName:='323 - Automaticky Rezim - model 5H, vymazanie vysledkov srobovania';
            SC_P1_Srobovanie.IdleTime.PT:= T#2s;
            SC_P1_Srobovanie.AlarmTime.PT:= T#5s;

            IF NOT SC_P1_Srobovanie.Switch1 THEN
                P1_Srobovanie.Skrutkovacka_K30.RESET_Vysledkov:= TRUE;
                SC_P1_Srobovanie.Switch1:= TRUE;
            END_IF

            IF NOT P1_Srobovanie.Skrutkovacka_K30.Stav_VysledokUtahovania_NG AND NOT P1_Srobovanie.Skrutkovacka_K30.Stav_VysledokUtahovania_OK AND NOT P1_Srobovanie.Skrutkovacka_K30.Stav_UtahovanieUkoncene THEN
                P1_Srobovanie.Skrutkovacka_K30.RESET_Vysledkov:= FALSE;
                SC_P1_Srobovanie.ResetStep:= TRUE;
                SC_P1_Srobovanie.Step:= 325;
            END_IF

        325:
            SC_P1_Srobovanie.StepName:='325 - Automaticky Rezim - model 5H, kontrola skrutky K30 v skrutkovacke';
            SC_P1_Srobovanie.IdleTime.PT:= T#5s;
            SC_P1_Srobovanie.AlarmTime.PT:= T#10s;
            SC_P1_Srobovanie.AlarmTime.IN:= TRUE;

            IF P1_Srobovanie.SkrutkovaciSet_K30.SkrutkaK30_Pripravena AND P1_Srobovanie.Skrutkovacka_K30.Stav_READY_to_START THEN
                SC_P1_Srobovanie.ResetStep:= TRUE;
                SC_P1_Srobovanie.Step:= 328;
            ELSIF SC_P1_Srobovanie.AlarmTime.Q THEN
                IF NOT P1_Srobovanie.Skrutkovacka_K30.Stav_READY_to_START THEN
                    P1_Alarmy[149]:= TRUE;
                    P1_StoperSrobovania.STAV.Porucha:= TRUE;
                    P1_Srobovanie.OUT.KOM_Srobovanie_Ukoncene:= TRUE;
                    SC_P1_Srobovanie.ResetStep:= TRUE;
                    SC_P1_Srobovanie.Step:= 338;
                ELSE
                    FazaNavratu:= 320;
                    SC_P1_Srobovanie.ResetStep:= TRUE;
                    SC_P1_Srobovanie.Step:= 500;
                END_IF
            END_IF

        328:
            SC_P1_Srobovanie.StepName:='328 - Automaticky Rezim - model 5H, vysunutie skrutkovacky K30';
            SC_P1_Srobovanie.IdleTime.PT:= T#2s;
            SC_P1_Srobovanie.AlarmTime.PT:= T#5s;

            SC_P1_Srobovanie.AlarmTime.IN:= (P1_Srobovanie.IN.SkrutkK30_VysunutieHrotu_IOS8 < 2);

            IF NOT SC_P1_Srobovanie.Switch1 THEN
                P1_Srobovanie.OUT.SkrutkK30_PrisavSkrutky_RUN_YV90:= TRUE;
                P1_Srobovanie.Skrutkovacka_K30.START_Utahovania:= TRUE;
                P1_Srobovanie.OUT.SkrutkK30_VYSUN_YV89:= TRUE;
                SC_P1_Srobovanie.Switch1:= TRUE;
            END_IF

            IF NOT P1_Srobovanie.Skrutkovacka_K30.Stav_UtahovanieUkoncene AND P1_Srobovanie.IN.SkrutkK30_VysunutieHrotu_IOS8 > 2 THEN
                SC_P1_Srobovanie.ResetStep:= TRUE;
                SC_P1_Srobovanie.Step:= 330;
            ELSIF SC_P1_Srobovanie.AlarmTime.Q THEN
                P1_Alarmy[142]:= TRUE;
                P1_Srobovanie.OUT.SkrutkK30_VYSUN_YV89:= FALSE;
                P1_Srobovanie.Skrutkovacka_K30.START_Utahovania:= FALSE;
                P1_StoperSrobovania.STAV.Porucha:= TRUE;
                P1_Srobovanie.OUT.KOM_Srobovanie_Ukoncene:= TRUE;
                SC_P1_Srobovanie.ResetStep:= TRUE;
                SC_P1_Srobovanie.Step:= 338;
            END_IF

        330:
            SC_P1_Srobovanie.StepName:='330 - Automaticky Rezim - model 5H, cakam na ukoncenie skrutkovania skrutkovacky K30';
            SC_P1_Srobovanie.IdleTime.PT:= T#30s;
            SC_P1_Srobovanie.AlarmTime.PT:= T#10s;
            SC_P1_Srobovanie.IdleTime.IN:= TRUE;
            SC_P1_Srobovanie.AlarmTime.IN:= TRUE;

            IF P1_Srobovanie.Skrutkovacka_K30.Stav_UtahovanieUkoncene THEN
                P1_Srobovanie.Skrutkovacka_K30.START_Utahovania:= FALSE;
                CasSrobovania:= TIME_TO_REAL(SC_P1_Srobovanie.IdleTime.ET);
                Reports.Skrutkovacky.VyskaSkrutkovania.P1_PravaSkrutkaK30:= REAL_TO_STRING(P1_Srobovanie.IN.SkrutkK30_VysunutieHrotu_IOS8);
                Reports.Skrutkovacky.CasSkrutkovania.P1_PravaSkrutkaK30:= REAL_TO_STRING(CasSrobovania/1000);
                SC_P1_Srobovanie.ResetStep:= TRUE;
                SC_P1_Srobovanie.Step:= 331;
            ELSIF SC_P1_Srobovanie.AlarmTime.Q THEN
                P1_Alarmy[146]:= TRUE;
                P1_Srobovanie.OUT.SkrutkK30_VYSUN_YV89:= FALSE;
                P1_Srobovanie.Skrutkovacka_K30.START_Utahovania:= FALSE;
                P1_StoperSrobovania.STAV.Porucha:= TRUE;
                P1_Srobovanie.OUT.KOM_Srobovanie_Ukoncene:= TRUE;
                SC_P1_Srobovanie.ResetStep:= TRUE;
                SC_P1_Srobovanie.Step:= 338;
            END_IF

        331:
            SC_P1_Srobovanie.StepName:='331 - Automaticky Rezim - model 5H, zasunutie skrutkovacky K30 a vypnutie prisavania skrutky';
            SC_P1_Srobovanie.IdleTime.PT:= T#200ms;
            SC_P1_Srobovanie.AlarmTime.PT:= T#5s;

            IF NOT SC_P1_Srobovanie.Switch1 THEN
                P1_Srobovanie.OUT.SkrutkK30_VYSUN_YV89:= FALSE;
                P1_Srobovanie.OUT.SkrutkK30_PrisavSkrutky_RUN_YV90:= FALSE;
                SC_P1_Srobovanie.Switch1:= TRUE;
            END_IF

            IF P1_Srobovanie.IN.SkrutkK30_ZASUNUTY_MS20 THEN
                SC_P1_Srobovanie.ResetStep:= TRUE;
                SC_P1_Srobovanie.Step:= 332;
            END_IF

        332:
            SC_P1_Srobovanie.StepName:='332 - Automaticky Rezim - model 5H, signal skrutka K30 odobrata';
            SC_P1_Srobovanie.IdleTime.PT:= T#200ms;
            SC_P1_Srobovanie.AlarmTime.PT:= T#5s;

            IF NOT SC_P1_Srobovanie.Switch1 THEN
                P1_Srobovanie.SkrutkovaciSet_K30.SkrutkaK30_Odobrata:= TRUE;
                SC_P1_Srobovanie.Switch1:= TRUE;
            END_IF

            IF NOT P1_Srobovanie.SkrutkovaciSet_K30.SkrutkaK30_Pripravena THEN
                P1_Srobovanie.SkrutkovaciSet_K30.SkrutkaK30_Odobrata:= FALSE;
                SC_P1_Srobovanie.ResetStep:= TRUE;
                SC_P1_Srobovanie.Step:= 335;
            END_IF

        335:
            SC_P1_Srobovanie.StepName:='335 - Automaticky Rezim - model 5H, kontrola vysledkov skrutkovania pravej skrutky K30';
            SC_P1_Srobovanie.IdleTime.PT:= T#200ms;
            SC_P1_Srobovanie.AlarmTime.PT:= T#5s;

            IF P1_Srobovanie.Skrutkovacka_K30.Stav_VysledokUtahovania_OK THEN
                P1_Srobovanie.STAV.Vysledok_Srobovania:= 'OK';
                P1_Srobovanie.OUT.KOM_Srobovanie_Ukoncene:= TRUE;
                SC_P1_Srobovanie.ResetStep:= TRUE;
                SC_P1_Srobovanie.Step:= 338;
            ELSIF P1_Srobovanie.Skrutkovacka_K30.Stav_VysledokUtahovania_NG THEN
                P1_Srobovanie.STAV.Vysledok_Srobovania:= 'NG';
                P1_Srobovanie.OUT.KOM_Srobovanie_Ukoncene:= TRUE;
                SC_P1_Srobovanie.ResetStep:= TRUE;
                SC_P1_Srobovanie.Step:= 338;
            END_IF

        338:
            SC_P1_Srobovanie.StepName:='338 - Automaticky Rezim - model 5H, cakam na zrusenie signalu zaskrutkuj pravu skrutku K30';
            SC_P1_Srobovanie.IdleTime.PT:= T#200ms;
            SC_P1_Srobovanie.AlarmTime.PT:= T#5s;

            IF NOT P1_StoperSrobovania.OUT.KOM_5H_ZasrobujPravuSkrutku_K30 THEN
                P1_Srobovanie.OUT.KOM_Srobovanie_Ukoncene:= FALSE;
                SC_P1_Srobovanie.ResetStep:= TRUE;
                SC_P1_Srobovanie.Step:= 100;
            END_IF

            //Zaskrutkovanie lavej skrutky M5//
        340:
            SC_P1_Srobovanie.StepName:='340 - Automaticky Rezim - model 5H, napolohovanie strednej skrutkovacky M5 na poziciu odobratia sroby M5 zo zasobnika';
            SC_P1_Srobovanie.IdleTime.PT:= T#200ms;
            SC_P1_Srobovanie.AlarmTime.PT:= T#5s;

            P1_Robot.KOM_OUT.ManipSrobovania_BezpecnaPozicia:= FALSE;

            P1_Srobovanie.PAR.OsX_ZadanaPozicia:= P1_RemPremenne.P1_Srob5H_PozX_OdobratSkrutkyM5; //mm
            P1_Srobovanie.PAR.OsY_ZadanaPozicia:= P1_RemPremenne.P1_Srob5H_PozY_OdobratSkrutkyM5; //mm

            IF NOT SC_P1_Srobovanie.Switch1 AND SC_OvlManipulatora_OsX.Step = 1 AND P1_Srobovacky_VychodziaPozicia AND Safety.STAV.P1_ZonaBunky_AKTIVNA THEN
                OsX_POLOHUJ:= TRUE;
                SC_P1_Srobovanie.Switch1:= TRUE;
            END_IF

            IF NOT SC_P1_Srobovanie.Switch2 AND SC_OvlManipulatora_OsY.Step = 1 AND P1_Srobovacky_VychodziaPozicia AND (P1_Srobovanie.ServoManipulOsX_M20.STATUS.ActualPosition > 14) AND Safety.STAV.P1_ZonaBunky_AKTIVNA THEN
                OsY_POLOHUJ:= TRUE;
                SC_P1_Srobovanie.Switch2:= TRUE;
            END_IF

            IF P1_Srobovanie.STAV.OsX_PoziciaDosiahnuta AND P1_Srobovanie.STAV.OsY_PoziciaDosiahnuta THEN
                P1_Srobovanie.STAV.OsX_PoziciaDosiahnuta:= FALSE;
                P1_Srobovanie.STAV.OsY_PoziciaDosiahnuta:= FALSE;
                IF P1_Srobovanie.RR_PolohujNaPoziciuSkrutky_5H THEN
                    P1_Srobovanie.RR_PolohujNaPoziciuSkrutky_5H:= FALSE;
                    P1_Srobovanie.RR_PolohujNaPoziciuSkrutky_4F:= FALSE;
                    P1_Srobovanie.RR_PolohujNaPoziciuSkrutky_5F:= FALSE;
                    SC_P1_Srobovanie.ResetStep:= TRUE;
                    SC_P1_Srobovanie.Step:= 700;
                ELSE
                    SC_P1_Srobovanie.ResetStep:= TRUE;
                    SC_P1_Srobovanie.Step:= 342;
                END_IF
            END_IF

        342:
            SC_P1_Srobovanie.StepName:='342 - Automaticky Rezim - model 5H, kontrola skrutky M5 na vystupe podavaca';
            SC_P1_Srobovanie.IdleTime.PT:= T#200ms;
            SC_P1_Srobovanie.AlarmTime.PT:= T#30s;
            SC_P1_Srobovanie.AlarmTime.IN:= TRUE;

            IF P1_Srobovanie.SkrutkovaciSet_M5.SkrutkaM5_Pripravena AND P1_Srobovanie.IN.OddelSrobM5_SrobaNaVystupe_OS14 THEN
                SC_P1_Srobovanie.ResetStep:= TRUE;
                SC_P1_Srobovanie.Step:= 343;
            ELSIF SC_P1_Srobovanie.AlarmTime.Q THEN
                P1_Alarmy[120]:= TRUE;
                P1_StoperSrobovania.STAV.Porucha:= TRUE;
                P1_Srobovanie.OUT.KOM_Srobovanie_Ukoncene:= TRUE;
                SC_P1_Srobovanie.ResetStep:= TRUE;
                SC_P1_Srobovanie.Step:= 353;
            END_IF

        343:
            SC_P1_Srobovanie.StepName:='343 - Automaticky Rezim - model 5H, odobratie skrutky M5 z podavaca';
            SC_P1_Srobovanie.IdleTime.PT:= T#200ms;
            SC_P1_Srobovanie.AlarmTime.PT:= T#5s;

            SC_P1_Srobovanie.IdleTime.IN:= P1_Srobovanie.IN.SkrutkM5_SnimacVakua_S28;

            IF NOT SC_P1_Srobovanie.Switch1 THEN
                P1_Srobovanie.OUT.SkrutkM5_VYSUN_YV104:= TRUE;
                P1_Srobovanie.OUT.SkrutkM5_PrisavSkrut_VYPNI_YV109:= FALSE;
                P1_Srobovanie.OUT.SkrutkM5_PrisavSkrut_ZAPNI_YV105:= TRUE;
                SC_P1_Srobovanie.IdleTime.IN:= TRUE;
                SC_P1_Srobovanie.Switch1:= TRUE;
            END_IF

            IF SC_P1_Srobovanie.IdleTime.Q THEN
                SC_P1_Srobovanie.ResetStep:= TRUE;
                SC_P1_Srobovanie.Step:= 344;
            END_IF

        344:
            SC_P1_Srobovanie.StepName:='344 - Automaticky Rezim - model 5H, zasunutie skrutkovacky M5, vystavenie signalu skrutka odobrata';
            SC_P1_Srobovanie.IdleTime.PT:= T#200ms;
            SC_P1_Srobovanie.AlarmTime.PT:= T#5s;

            IF NOT SC_P1_Srobovanie.Switch1 THEN
                P1_Srobovanie.OUT.SkrutkM5_VYSUN_YV104:= FALSE;
                SC_P1_Srobovanie.Switch1:= TRUE;
            END_IF

            IF P1_Srobovanie.IN.SkrutkM5_ZASUNUTY_MS39 THEN
                P1_Srobovanie.SkrutkovaciSet_M5.SkrutkaM5_Odobrata:= TRUE;
                SC_P1_Srobovanie.ResetStep:= TRUE;
                SC_P1_Srobovanie.Step:= 345;
            END_IF

        345:
            SC_P1_Srobovanie.StepName:='345 - Automaticky Rezim - model 5H, cakam na zrusenie signalu skrutka M5 pripravena';
            SC_P1_Srobovanie.IdleTime.PT:= T#200ms;
            SC_P1_Srobovanie.AlarmTime.PT:= T#5s;

            IF NOT P1_Srobovanie.SkrutkovaciSet_M5.SkrutkaM5_Pripravena THEN
                P1_Srobovanie.SkrutkovaciSet_M5.SkrutkaM5_Odobrata:= FALSE;
                SC_P1_Srobovanie.ResetStep:= TRUE;
                SC_P1_Srobovanie.Step:= 346;
            END_IF

        346:
            SC_P1_Srobovanie.StepName:='346 - Automaticky Rezim - model 5H, napolohovanie strednej skrutkovacky M5 na poziciu lavej skrutky M5';
            SC_P1_Srobovanie.IdleTime.PT:= T#200ms;
            SC_P1_Srobovanie.AlarmTime.PT:= T#5s;

            P1_Robot.KOM_OUT.ManipSrobovania_BezpecnaPozicia:= FALSE;

            P1_Srobovanie.PAR.OsX_ZadanaPozicia:= P1_RemPremenne.P1_Srob5H_PozX_LavejSkrutkyM5; //mm
            P1_Srobovanie.PAR.OsY_ZadanaPozicia:= P1_RemPremenne.P1_Srob5H_PozY_LavejSkrutkyM5; //mm

            IF NOT SC_P1_Srobovanie.Switch1 AND SC_OvlManipulatora_OsX.Step = 1 AND P1_Srobovacky_VychodziaPozicia AND Safety.STAV.P1_ZonaBunky_AKTIVNA THEN
                OsX_POLOHUJ:= TRUE;
                SC_P1_Srobovanie.Switch1:= TRUE;
            END_IF

            IF NOT SC_P1_Srobovanie.Switch2 AND SC_OvlManipulatora_OsY.Step = 1 AND P1_Srobovacky_VychodziaPozicia AND (P1_Srobovanie.ServoManipulOsX_M20.STATUS.ActualPosition > 14) AND Safety.STAV.P1_ZonaBunky_AKTIVNA THEN
                OsY_POLOHUJ:= TRUE;
                SC_P1_Srobovanie.Switch2:= TRUE;
            END_IF

            IF P1_Srobovanie.STAV.OsX_PoziciaDosiahnuta AND P1_Srobovanie.STAV.OsY_PoziciaDosiahnuta THEN
                P1_Srobovanie.STAV.OsX_PoziciaDosiahnuta:= FALSE;
                P1_Srobovanie.STAV.OsY_PoziciaDosiahnuta:= FALSE;
                IF P1_Srobovanie.RR_PolohujNaPoziciuSkrutky_5H THEN
                    P1_Srobovanie.RR_PolohujNaPoziciuSkrutky_5H:= FALSE;
                    P1_Srobovanie.RR_PolohujNaPoziciuSkrutky_4F:= FALSE;
                    P1_Srobovanie.RR_PolohujNaPoziciuSkrutky_5F:= FALSE;
                    SC_P1_Srobovanie.ResetStep:= TRUE;
                    SC_P1_Srobovanie.Step:= 700;
                ELSE
                    SC_P1_Srobovanie.ResetStep:= TRUE;
                    SC_P1_Srobovanie.Step:= 347;
                END_IF
            END_IF

        347:
            SC_P1_Srobovanie.StepName:='347 - Automaticky Rezim - model 5H, vymazanie vysledkov srobovania, prepnutie programu';
            SC_P1_Srobovanie.IdleTime.PT:= T#2s;
            SC_P1_Srobovanie.AlarmTime.PT:= T#5s;

            IF NOT SC_P1_Srobovanie.Switch1 THEN
                P1_Srobovanie.Skrutkovacka_M5.RESET_Vysledkov:= TRUE;
                SC_P1_Srobovanie.Switch1:= TRUE;
            END_IF

            IF NOT P1_Srobovanie.Skrutkovacka_M5.Stav_VysledokUtahovania_NG AND NOT P1_Srobovanie.Skrutkovacka_M5.Stav_VysledokUtahovania_OK THEN
                P1_Srobovanie.Skrutkovacka_M5.RESET_Vysledkov:= FALSE;
                SC_P1_Srobovanie.ResetStep:= TRUE;
                SC_P1_Srobovanie.Step:= 348;
            END_IF

        348:
            SC_P1_Srobovanie.StepName:='348 - Automaticky Rezim - model 5H, prepnutie programu a kontrola skrutkovacky';
            SC_P1_Srobovanie.IdleTime.PT:= T#2s;
            SC_P1_Srobovanie.AlarmTime.PT:= T#10s;

            IF NOT SC_P1_Srobovanie.Switch1 THEN
                P1_Srobovanie.Skrutkovacka_M5.CisloZadanehoProgramu:= 2;
                SC_P1_Srobovanie.AlarmTime.IN:= TRUE;
                SC_P1_Srobovanie.Switch1:= TRUE;
            END_IF

            IF P1_Srobovanie.Skrutkovacka_M5.Stav_CisloAktualnehoProgramu = 2 AND P1_Srobovanie.Skrutkovacka_M5.Stav_READY_to_START AND NOT P1_Srobovanie.Skrutkovacka_M5.Stav_UtahovanieUkoncene THEN
                SC_P1_Srobovanie.ResetStep:= TRUE;
                SC_P1_Srobovanie.Step:= 349;
            ELSIF SC_P1_Srobovanie.AlarmTime.Q AND NOT P1_Srobovanie.Skrutkovacka_M5.Stav_READY_to_START THEN
                P1_Alarmy[150]:= TRUE;
                P1_StoperSrobovania.STAV.Porucha:= TRUE;
                P1_Srobovanie.OUT.KOM_Srobovanie_Ukoncene:= TRUE;
                SC_P1_Srobovanie.ResetStep:= TRUE;
                SC_P1_Srobovanie.Step:= 353;
            END_IF

        349:
            SC_P1_Srobovanie.StepName:='349 - Automaticky Rezim - model 5H, vysunutie skrutkovacky M5';
            SC_P1_Srobovanie.IdleTime.PT:= T#2s;
            SC_P1_Srobovanie.AlarmTime.PT:= T#5s;

            SC_P1_Srobovanie.AlarmTime.IN:= (P1_Srobovanie.IN.SkrutkM5_VysunutieHrotu_IOS9 < 2);

            IF NOT SC_P1_Srobovanie.Switch1 THEN
                P1_Srobovanie.OUT.SkrutkM5_VYSUN_YV104:= TRUE;
                P1_Srobovanie.Skrutkovacka_M5.START_Utahovania:= TRUE;
                SC_P1_Srobovanie.Switch1:= TRUE;
            END_IF

            IF NOT P1_Srobovanie.Skrutkovacka_M5.Stav_UtahovanieUkoncene AND P1_Srobovanie.IN.SkrutkM5_VysunutieHrotu_IOS9 > 2 AND NOT TEST THEN
                SC_P1_Srobovanie.ResetStep:= TRUE;
                SC_P1_Srobovanie.Step:= 350;
            ELSIF SC_P1_Srobovanie.AlarmTime.Q AND NOT TEST THEN
                P1_Alarmy[143]:= TRUE;
                P1_Srobovanie.OUT.SkrutkM5_VYSUN_YV104:= FALSE;
                P1_Srobovanie.Skrutkovacka_M5.START_Utahovania:= FALSE;
                P1_StoperSrobovania.STAV.Porucha:= TRUE;
                P1_Srobovanie.OUT.KOM_Srobovanie_Ukoncene:= TRUE;
                SC_P1_Srobovanie.ResetStep:= TRUE;
                SC_P1_Srobovanie.Step:= 353;
            END_IF

        350:
            SC_P1_Srobovanie.StepName:='350 - Automaticky Rezim - model 5H, cakam na ukoncenie skrutkovania skrutkovacky M5';
            SC_P1_Srobovanie.IdleTime.PT:= T#30s;
            SC_P1_Srobovanie.AlarmTime.PT:= T#10s;
            SC_P1_Srobovanie.IdleTime.IN:= TRUE;
            SC_P1_Srobovanie.AlarmTime.IN:= TRUE;

            IF P1_Srobovanie.Skrutkovacka_M5.Stav_UtahovanieUkoncene THEN
                P1_Srobovanie.Skrutkovacka_M5.START_Utahovania:= FALSE;
                CasSrobovania:= TIME_TO_REAL(SC_P1_Srobovanie.IdleTime.ET);
                Reports.Skrutkovacky.VyskaSkrutkovania.P1_LavaSkrutkaM5:= REAL_TO_STRING(P1_Srobovanie.IN.SkrutkM5_VysunutieHrotu_IOS9);
                Reports.Skrutkovacky.CasSkrutkovania.P1_LavaSkrutkaM5:= REAL_TO_STRING(CasSrobovania/1000);
                SC_P1_Srobovanie.ResetStep:= TRUE;
                SC_P1_Srobovanie.Step:= 351;
            ELSIF SC_P1_Srobovanie.AlarmTime.Q THEN
                P1_Alarmy[147]:= TRUE;
                P1_Srobovanie.OUT.SkrutkM5_VYSUN_YV104:= FALSE;
                P1_Srobovanie.Skrutkovacka_M5.START_Utahovania:= FALSE;
                P1_StoperSrobovania.STAV.Porucha:= TRUE;
                P1_Srobovanie.OUT.KOM_Srobovanie_Ukoncene:= TRUE;
                SC_P1_Srobovanie.ResetStep:= TRUE;
                SC_P1_Srobovanie.Step:= 353;
            END_IF

        351:
            SC_P1_Srobovanie.StepName:='351 - Automaticky Rezim - model 5H, zasunutie skrutkovacky M5 a vypnutie prisavania skrutky';
            SC_P1_Srobovanie.IdleTime.PT:= T#200ms;
            SC_P1_Srobovanie.AlarmTime.PT:= T#5s;

            IF NOT SC_P1_Srobovanie.Switch1 THEN
                P1_Srobovanie.OUT.SkrutkM5_VYSUN_YV104:= FALSE;
                P1_Srobovanie.OUT.SkrutkM5_PrisavSkrut_ZAPNI_YV105:= FALSE;
                P1_Srobovanie.OUT.SkrutkM5_PrisavSkrut_VYPNI_YV109:= TRUE;
                SC_P1_Srobovanie.Switch1:= TRUE;
            END_IF

            IF P1_Srobovanie.IN.SkrutkM5_ZASUNUTY_MS39 THEN
                SC_P1_Srobovanie.ResetStep:= TRUE;
                SC_P1_Srobovanie.Step:= 352;
            END_IF

        352:
            SC_P1_Srobovanie.StepName:='352 - Automaticky Rezim - model 5H, kontrola vysledkov skrutkovania lavej skrutky M5';
            SC_P1_Srobovanie.IdleTime.PT:= T#200ms;
            SC_P1_Srobovanie.AlarmTime.PT:= T#5s;

            IF P1_Srobovanie.Skrutkovacka_M5.Stav_VysledokUtahovania_OK THEN
                P1_Srobovanie.STAV.Vysledok_Srobovania:= 'OK';
                P1_Srobovanie.OUT.KOM_Srobovanie_Ukoncene:= TRUE;
                SC_P1_Srobovanie.ResetStep:= TRUE;
                SC_P1_Srobovanie.Step:= 353;
            ELSIF P1_Srobovanie.Skrutkovacka_M5.Stav_VysledokUtahovania_NG THEN
                P1_Srobovanie.STAV.Vysledok_Srobovania:= 'NG';
                P1_Srobovanie.OUT.KOM_Srobovanie_Ukoncene:= TRUE;
                SC_P1_Srobovanie.ResetStep:= TRUE;
                SC_P1_Srobovanie.Step:= 353;
            END_IF

        353:
            SC_P1_Srobovanie.StepName:='353 - Automaticky Rezim - model 5H, cakam na zrusenie signalu zaskrutkuj lavu skrutku M5';
            SC_P1_Srobovanie.IdleTime.PT:= T#200ms;
            SC_P1_Srobovanie.AlarmTime.PT:= T#5s;

            IF NOT P1_StoperSrobovania.OUT.KOM_5H_ZasrobujLavuSkrutku_M5 THEN
                P1_Srobovanie.OUT.KOM_Srobovanie_Ukoncene:= FALSE;
                SC_P1_Srobovanie.ResetStep:= TRUE;
                SC_P1_Srobovanie.Step:= 100;
            END_IF

            //Zaskrutkovanie pravej skrutky M5//
        360:
            SC_P1_Srobovanie.StepName:='360 - Automaticky Rezim - model 5H, napolohovanie strednej skrutkovacky M5 na poziciu odobratia sroby M5 zo zasobnika';
            SC_P1_Srobovanie.IdleTime.PT:= T#200ms;
            SC_P1_Srobovanie.AlarmTime.PT:= T#5s;

            P1_Robot.KOM_OUT.ManipSrobovania_BezpecnaPozicia:= FALSE;

            P1_Srobovanie.PAR.OsX_ZadanaPozicia:= P1_RemPremenne.P1_Srob5H_PozX_OdobratSkrutkyM5; //mm
            P1_Srobovanie.PAR.OsY_ZadanaPozicia:= P1_RemPremenne.P1_Srob5H_PozY_OdobratSkrutkyM5; //mm

            IF NOT SC_P1_Srobovanie.Switch1 AND SC_OvlManipulatora_OsX.Step = 1 AND P1_Srobovacky_VychodziaPozicia AND Safety.STAV.P1_ZonaBunky_AKTIVNA THEN
                OsX_POLOHUJ:= TRUE;
                SC_P1_Srobovanie.Switch1:= TRUE;
            END_IF

            IF NOT SC_P1_Srobovanie.Switch2 AND SC_OvlManipulatora_OsY.Step = 1 AND P1_Srobovacky_VychodziaPozicia AND (P1_Srobovanie.ServoManipulOsX_M20.STATUS.ActualPosition > 14) AND Safety.STAV.P1_ZonaBunky_AKTIVNA THEN
                OsY_POLOHUJ:= TRUE;
                SC_P1_Srobovanie.Switch2:= TRUE;
            END_IF

            IF P1_Srobovanie.STAV.OsX_PoziciaDosiahnuta AND P1_Srobovanie.STAV.OsY_PoziciaDosiahnuta THEN
                P1_Srobovanie.STAV.OsX_PoziciaDosiahnuta:= FALSE;
                P1_Srobovanie.STAV.OsY_PoziciaDosiahnuta:= FALSE;
                SC_P1_Srobovanie.ResetStep:= TRUE;
                SC_P1_Srobovanie.Step:= 361;
            END_IF

        361:
            SC_P1_Srobovanie.StepName:='361 - Automaticky Rezim - model 5H, kontrola skrutky M5 na vystupe podavaca';
            SC_P1_Srobovanie.IdleTime.PT:= T#200ms;
            SC_P1_Srobovanie.AlarmTime.PT:= T#30s;
            SC_P1_Srobovanie.AlarmTime.IN:= TRUE;

            IF P1_Srobovanie.SkrutkovaciSet_M5.SkrutkaM5_Pripravena AND P1_Srobovanie.IN.OddelSrobM5_SrobaNaVystupe_OS14 THEN
                SC_P1_Srobovanie.ResetStep:= TRUE;
                SC_P1_Srobovanie.Step:= 362;
            ELSIF SC_P1_Srobovanie.AlarmTime.Q THEN
                P1_Alarmy[120]:= TRUE;
                P1_StoperSrobovania.STAV.Porucha:= TRUE;
                P1_Srobovanie.OUT.KOM_Srobovanie_Ukoncene:= TRUE;
                SC_P1_Srobovanie.ResetStep:= TRUE;
                SC_P1_Srobovanie.Step:= 378;
            END_IF

        362:
            SC_P1_Srobovanie.StepName:='362 - Automaticky Rezim - model 5H, odobratie skrutky M5 z podavaca';
            SC_P1_Srobovanie.IdleTime.PT:= T#200ms;
            SC_P1_Srobovanie.AlarmTime.PT:= T#5s;

            SC_P1_Srobovanie.IdleTime.IN:= P1_Srobovanie.IN.SkrutkM5_SnimacVakua_S28;

            IF NOT SC_P1_Srobovanie.Switch1 THEN
                P1_Srobovanie.OUT.SkrutkM5_VYSUN_YV104:= TRUE;
                P1_Srobovanie.OUT.SkrutkM5_PrisavSkrut_VYPNI_YV109:= FALSE;
                P1_Srobovanie.OUT.SkrutkM5_PrisavSkrut_ZAPNI_YV105:= TRUE;
                SC_P1_Srobovanie.IdleTime.IN:= TRUE;
                SC_P1_Srobovanie.Switch1:= TRUE;
            END_IF

            IF SC_P1_Srobovanie.IdleTime.Q THEN
                SC_P1_Srobovanie.ResetStep:= TRUE;
                SC_P1_Srobovanie.Step:= 363;
            END_IF

        363:
            SC_P1_Srobovanie.StepName:='363 - Automaticky Rezim - model 5H, zasunutie skrutkovacky M5, vystavenie signalu skrutka odobrata';
            SC_P1_Srobovanie.IdleTime.PT:= T#200ms;
            SC_P1_Srobovanie.AlarmTime.PT:= T#5s;

            IF NOT SC_P1_Srobovanie.Switch1 THEN
                P1_Srobovanie.OUT.SkrutkM5_VYSUN_YV104:= FALSE;
                SC_P1_Srobovanie.Switch1:= TRUE;
            END_IF

            IF P1_Srobovanie.IN.SkrutkM5_ZASUNUTY_MS39 THEN
                P1_Srobovanie.SkrutkovaciSet_M5.SkrutkaM5_Odobrata:= TRUE;
                SC_P1_Srobovanie.ResetStep:= TRUE;
                SC_P1_Srobovanie.Step:= 364;
            END_IF

        364:
            SC_P1_Srobovanie.StepName:='364 - Automaticky Rezim - model 5H, cakam na zrusenie signalu skrutka M5 pripravena';
            SC_P1_Srobovanie.IdleTime.PT:= T#200ms;
            SC_P1_Srobovanie.AlarmTime.PT:= T#5s;

            IF NOT P1_Srobovanie.SkrutkovaciSet_M5.SkrutkaM5_Pripravena THEN
                P1_Srobovanie.SkrutkovaciSet_M5.SkrutkaM5_Odobrata:= FALSE;
                SC_P1_Srobovanie.ResetStep:= TRUE;
                SC_P1_Srobovanie.Step:= 366;
            END_IF

        365:
            SC_P1_Srobovanie.StepName:='365 - Automaticky Rezim - model 5H, napolohovanie strednej skrutkovacky M5 na poziciu strednej skrutky M5';
            SC_P1_Srobovanie.IdleTime.PT:= T#200ms;
            SC_P1_Srobovanie.AlarmTime.PT:= T#5s;

            P1_Robot.KOM_OUT.ManipSrobovania_BezpecnaPozicia:= FALSE;

            P1_Srobovanie.PAR.OsX_ZadanaPozicia:= P1_RemPremenne.P1_Srob5H_PozX_StrednejSkrutkyM5; //mm
            P1_Srobovanie.PAR.OsY_ZadanaPozicia:= P1_RemPremenne.P1_Srob5H_PozY_StrednejSkrutkyM5; //mm

            IF NOT SC_P1_Srobovanie.Switch1 AND SC_OvlManipulatora_OsX.Step = 1 AND P1_Srobovacky_VychodziaPozicia AND Safety.STAV.P1_ZonaBunky_AKTIVNA THEN
                OsX_POLOHUJ:= TRUE;
                SC_P1_Srobovanie.Switch1:= TRUE;
            END_IF

            IF NOT SC_P1_Srobovanie.Switch2 AND SC_OvlManipulatora_OsY.Step = 1 AND P1_Srobovacky_VychodziaPozicia AND (P1_Srobovanie.ServoManipulOsX_M20.STATUS.ActualPosition > 14) AND Safety.STAV.P1_ZonaBunky_AKTIVNA THEN
                OsY_POLOHUJ:= TRUE;
                SC_P1_Srobovanie.Switch2:= TRUE;
            END_IF

            IF P1_Srobovanie.STAV.OsX_PoziciaDosiahnuta AND P1_Srobovanie.STAV.OsY_PoziciaDosiahnuta THEN
                P1_Srobovanie.STAV.OsX_PoziciaDosiahnuta:= FALSE;
                P1_Srobovanie.STAV.OsY_PoziciaDosiahnuta:= FALSE;
                SC_P1_Srobovanie.ResetStep:= TRUE;
                SC_P1_Srobovanie.Step:= 366;
            END_IF

        366:
            SC_P1_Srobovanie.StepName:='366 - Automaticky Rezim - model 5H, napolohovanie strednej skrutkovacky M5 na poziciu pravej skrutky M5';
            SC_P1_Srobovanie.IdleTime.PT:= T#200ms;
            SC_P1_Srobovanie.AlarmTime.PT:= T#5s;

            P1_Robot.KOM_OUT.ManipSrobovania_BezpecnaPozicia:= FALSE;

            P1_Srobovanie.PAR.OsX_ZadanaPozicia:= P1_RemPremenne.P1_Srob5H_PozX_PravejSkrutkyM5; //mm
            P1_Srobovanie.PAR.OsY_ZadanaPozicia:= P1_RemPremenne.P1_Srob5H_PozY_PravejSkrutkyM5; //mm

            IF NOT SC_P1_Srobovanie.Switch1 AND SC_OvlManipulatora_OsY.Step = 1 AND P1_Srobovacky_VychodziaPozicia AND Safety.STAV.P1_ZonaBunky_AKTIVNA THEN
                OsY_POLOHUJ:= TRUE;
                SC_P1_Srobovanie.Switch1:= TRUE;
            END_IF

            IF NOT SC_P1_Srobovanie.Switch2 AND SC_OvlManipulatora_OsX.Step = 1 AND P1_Srobovacky_VychodziaPozicia AND (P1_Srobovanie.ServoManipulOsY_M19.STATUS.ActualPosition > 240) AND Safety.STAV.P1_ZonaBunky_AKTIVNA THEN
                OsX_POLOHUJ:= TRUE;
                SC_P1_Srobovanie.Switch2:= TRUE;
            END_IF

            IF P1_Srobovanie.STAV.OsX_PoziciaDosiahnuta AND P1_Srobovanie.STAV.OsY_PoziciaDosiahnuta THEN
                P1_Srobovanie.STAV.OsX_PoziciaDosiahnuta:= FALSE;
                P1_Srobovanie.STAV.OsY_PoziciaDosiahnuta:= FALSE;
                IF P1_Srobovanie.RR_PolohujNaPoziciuSkrutky_5H THEN
                    P1_Srobovanie.RR_PolohujNaPoziciuSkrutky_5H:= FALSE;
                    P1_Srobovanie.RR_PolohujNaPoziciuSkrutky_4F:= FALSE;
                    P1_Srobovanie.RR_PolohujNaPoziciuSkrutky_5F:= FALSE;
                    SC_P1_Srobovanie.ResetStep:= TRUE;
                    SC_P1_Srobovanie.Step:= 700;
                ELSE
                    SC_P1_Srobovanie.ResetStep:= TRUE;
                    SC_P1_Srobovanie.Step:= 367;
                END_IF
            END_IF

        367:
            SC_P1_Srobovanie.StepName:='367 - Automaticky Rezim - model 5H, vymazanie vysledkov srobovania';
            SC_P1_Srobovanie.IdleTime.PT:= T#2s;
            SC_P1_Srobovanie.AlarmTime.PT:= T#5s;

            IF NOT SC_P1_Srobovanie.Switch1 THEN
                P1_Srobovanie.Skrutkovacka_M5.RESET_Vysledkov:= TRUE;
                SC_P1_Srobovanie.Switch1:= TRUE;
            END_IF

            IF NOT P1_Srobovanie.Skrutkovacka_M5.Stav_VysledokUtahovania_NG AND NOT P1_Srobovanie.Skrutkovacka_M5.Stav_VysledokUtahovania_OK THEN
                P1_Srobovanie.Skrutkovacka_M5.RESET_Vysledkov:= FALSE;
                SC_P1_Srobovanie.ResetStep:= TRUE;
                SC_P1_Srobovanie.Step:= 368;
            END_IF

        368:
            SC_P1_Srobovanie.StepName:='368 - Automaticky Rezim - model 5H, prepnutie programu a kontrola stavu skrutkovacky';
            SC_P1_Srobovanie.IdleTime.PT:= T#2s;
            SC_P1_Srobovanie.AlarmTime.PT:= T#10s;

            IF NOT SC_P1_Srobovanie.Switch1 THEN
                P1_Srobovanie.Skrutkovacka_M5.CisloZadanehoProgramu:= 2;
                SC_P1_Srobovanie.AlarmTime.IN:= TRUE;
                SC_P1_Srobovanie.Switch1:= TRUE;
            END_IF

            IF P1_Srobovanie.Skrutkovacka_M5.Stav_CisloAktualnehoProgramu = 2 AND P1_Srobovanie.Skrutkovacka_M5.Stav_READY_to_START AND NOT P1_Srobovanie.Skrutkovacka_M5.Stav_UtahovanieUkoncene THEN
                SC_P1_Srobovanie.ResetStep:= TRUE;
                SC_P1_Srobovanie.Step:= 370;
            ELSIF SC_P1_Srobovanie.AlarmTime.Q AND NOT P1_Srobovanie.Skrutkovacka_M5.Stav_READY_to_START THEN
                P1_Alarmy[150]:= TRUE;
                P1_StoperSrobovania.STAV.Porucha:= TRUE;
                P1_Srobovanie.OUT.KOM_Srobovanie_Ukoncene:= TRUE;
                SC_P1_Srobovanie.ResetStep:= TRUE;
                SC_P1_Srobovanie.Step:= 378;
            END_IF

        370:
            SC_P1_Srobovanie.StepName:='370 - Automaticky Rezim - model 5H, vysunutie skrutkovacky M5';
            SC_P1_Srobovanie.IdleTime.PT:= T#2s;
            SC_P1_Srobovanie.AlarmTime.PT:= T#5s;

            SC_P1_Srobovanie.AlarmTime.IN:= (P1_Srobovanie.IN.SkrutkM5_VysunutieHrotu_IOS9 < 2);

            IF NOT SC_P1_Srobovanie.Switch1 THEN
                P1_Srobovanie.OUT.SkrutkM5_VYSUN_YV104:= TRUE;
                P1_Srobovanie.Skrutkovacka_M5.START_Utahovania:= TRUE;
                SC_P1_Srobovanie.Switch1:= TRUE;
            END_IF

            IF NOT P1_Srobovanie.Skrutkovacka_M5.Stav_UtahovanieUkoncene AND P1_Srobovanie.IN.SkrutkM5_VysunutieHrotu_IOS9 > 2 THEN
                SC_P1_Srobovanie.ResetStep:= TRUE;
                SC_P1_Srobovanie.Step:= 371;
            ELSIF SC_P1_Srobovanie.AlarmTime.Q THEN
                P1_Alarmy[143]:= TRUE;
                P1_Srobovanie.OUT.SkrutkM5_VYSUN_YV104:= FALSE;
                P1_Srobovanie.Skrutkovacka_M5.START_Utahovania:= FALSE;
                P1_StoperSrobovania.STAV.Porucha:= TRUE;
                P1_Srobovanie.OUT.KOM_Srobovanie_Ukoncene:= TRUE;
                SC_P1_Srobovanie.ResetStep:= TRUE;
                SC_P1_Srobovanie.Step:= 378;
            END_IF

        371:
            SC_P1_Srobovanie.StepName:='371 - Automaticky Rezim - model 5H, cakam na ukoncenie skrutkovania skrutkovacky M5';
            SC_P1_Srobovanie.IdleTime.PT:= T#30s;
            SC_P1_Srobovanie.AlarmTime.PT:= T#10s;
            SC_P1_Srobovanie.IdleTime.IN:= TRUE;
            SC_P1_Srobovanie.AlarmTime.IN:= TRUE;

            IF P1_Srobovanie.Skrutkovacka_M5.Stav_UtahovanieUkoncene THEN
                P1_Srobovanie.Skrutkovacka_M5.START_Utahovania:= FALSE;
                CasSrobovania:= TIME_TO_REAL(SC_P1_Srobovanie.IdleTime.ET);
                Reports.Skrutkovacky.VyskaSkrutkovania.P1_PravaSkrutkaM5:= REAL_TO_STRING(P1_Srobovanie.IN.SkrutkM5_VysunutieHrotu_IOS9);
                Reports.Skrutkovacky.CasSkrutkovania.P1_PravaSkrutkaM5:= REAL_TO_STRING(CasSrobovania/1000);
                SC_P1_Srobovanie.ResetStep:= TRUE;
                SC_P1_Srobovanie.Step:= 373;
            ELSIF SC_P1_Srobovanie.AlarmTime.Q THEN
                P1_Alarmy[147]:= TRUE;
                P1_Srobovanie.OUT.SkrutkM5_VYSUN_YV104:= FALSE;
                P1_Srobovanie.Skrutkovacka_M5.START_Utahovania:= FALSE;
                P1_StoperSrobovania.STAV.Porucha:= TRUE;
                P1_Srobovanie.OUT.KOM_Srobovanie_Ukoncene:= TRUE;
                SC_P1_Srobovanie.ResetStep:= TRUE;
                SC_P1_Srobovanie.Step:= 378;
            END_IF

        373:
            SC_P1_Srobovanie.StepName:='373 - Automaticky Rezim - model 5H, vystavenie signalu pre robota uvolni busbary';
            SC_P1_Srobovanie.IdleTime.PT:= T#30s;
            SC_P1_Srobovanie.AlarmTime.PT:= T#10s;

            IF NOT SC_P1_Srobovanie.Switch1 THEN
                P1_Robot.KOM_OUT.UvolniBusbary:= TRUE;
                SC_P1_Srobovanie.Switch1:= TRUE;
            END_IF

            IF P1_Robot.KOM_IN.Stav_BusbaryUvolnene THEN
                P1_Robot.KOM_OUT.UvolniBusbary:= FALSE;
                SC_P1_Srobovanie.ResetStep:= TRUE;
                SC_P1_Srobovanie.Step:= 374;
            END_IF

        374:
            SC_P1_Srobovanie.StepName:='374 - Automaticky Rezim - model 5H, zasunutie skrutkovacky M5 a vypnutie prisavania skrutky';
            SC_P1_Srobovanie.IdleTime.PT:= T#200ms;
            SC_P1_Srobovanie.AlarmTime.PT:= T#5s;

            IF NOT SC_P1_Srobovanie.Switch1 AND NOT P1_Robot.KOM_IN.Stav_BusbaryUvolnene THEN
                P1_Srobovanie.OUT.SkrutkM5_VYSUN_YV104:= FALSE;
                P1_Srobovanie.OUT.SkrutkM5_PrisavSkrut_ZAPNI_YV105:= FALSE;
                P1_Srobovanie.OUT.SkrutkM5_PrisavSkrut_VYPNI_YV109:= TRUE;
                SC_P1_Srobovanie.Switch1:= TRUE;
            END_IF

            IF P1_Srobovanie.IN.SkrutkM5_ZASUNUTY_MS39 THEN
                SC_P1_Srobovanie.ResetStep:= TRUE;
                SC_P1_Srobovanie.Step:= 375;
            END_IF

        375:
            SC_P1_Srobovanie.StepName:='375 - Automaticky Rezim - model 5H, kontrola vysledkov skrutkovania pravej skrutky M5';
            SC_P1_Srobovanie.IdleTime.PT:= T#200ms;
            SC_P1_Srobovanie.AlarmTime.PT:= T#5s;

            IF P1_Srobovanie.Skrutkovacka_M5.Stav_VysledokUtahovania_OK THEN
                P1_Srobovanie.STAV.Vysledok_Srobovania:= 'OK';
                P1_Srobovanie.OUT.KOM_Srobovanie_Ukoncene:= TRUE;
                SC_P1_Srobovanie.ResetStep:= TRUE;
                SC_P1_Srobovanie.Step:= 376;
            ELSIF P1_Srobovanie.Skrutkovacka_M5.Stav_VysledokUtahovania_NG THEN
                P1_Srobovanie.STAV.Vysledok_Srobovania:= 'NG';
                P1_Srobovanie.OUT.KOM_Srobovanie_Ukoncene:= TRUE;
                SC_P1_Srobovanie.ResetStep:= TRUE;
                SC_P1_Srobovanie.Step:= 376;
            END_IF

        376:
            SC_P1_Srobovanie.StepName:='376 - Automaticky Rezim - model 5H, napolohovanie strednej skrutkovacky M5 na poziciu strednej skrutky M5';
            SC_P1_Srobovanie.IdleTime.PT:= T#200ms;
            SC_P1_Srobovanie.AlarmTime.PT:= T#5s;

            P1_Robot.KOM_OUT.ManipSrobovania_BezpecnaPozicia:= FALSE;

            P1_Srobovanie.PAR.OsX_ZadanaPozicia:= P1_RemPremenne.P1_Srob5H_PozX_StrednejSkrutkyM5; //mm
            P1_Srobovanie.PAR.OsY_ZadanaPozicia:= P1_RemPremenne.P1_Srob5H_PozY_StrednejSkrutkyM5; //mm

            IF NOT SC_P1_Srobovanie.Switch1 AND SC_OvlManipulatora_OsX.Step = 1 AND P1_Srobovacky_VychodziaPozicia AND Safety.STAV.P1_ZonaBunky_AKTIVNA THEN
                OsX_POLOHUJ:= TRUE;
                SC_P1_Srobovanie.Switch1:= TRUE;
            END_IF

            IF NOT SC_P1_Srobovanie.Switch2 AND SC_OvlManipulatora_OsY.Step = 1 AND P1_Srobovacky_VychodziaPozicia AND (P1_Srobovanie.ServoManipulOsX_M20.STATUS.ActualPosition > 14) AND Safety.STAV.P1_ZonaBunky_AKTIVNA THEN
                OsY_POLOHUJ:= TRUE;
                SC_P1_Srobovanie.Switch2:= TRUE;
            END_IF

            IF P1_Srobovanie.STAV.OsX_PoziciaDosiahnuta AND P1_Srobovanie.STAV.OsY_PoziciaDosiahnuta THEN
                P1_Srobovanie.STAV.OsX_PoziciaDosiahnuta:= FALSE;
                P1_Srobovanie.STAV.OsY_PoziciaDosiahnuta:= FALSE;
                SC_P1_Srobovanie.ResetStep:= TRUE;
                SC_P1_Srobovanie.Step:= 378;
            END_IF

        378:
            SC_P1_Srobovanie.StepName:='378 - Automaticky Rezim - model 5H, cakam na zrusenie signalu zaskrutkuj pravu skrutku M5';
            SC_P1_Srobovanie.IdleTime.PT:= T#200ms;
            SC_P1_Srobovanie.AlarmTime.PT:= T#5s;

            IF NOT P1_StoperSrobovania.OUT.KOM_5H_ZasrobujPravuSkrutku_M5 THEN
                P1_Srobovanie.OUT.KOM_Srobovanie_Ukoncene:= FALSE;
                SC_P1_Srobovanie.ResetStep:= TRUE;
                SC_P1_Srobovanie.Step:= 100;
            END_IF

            //Zaskrutkovanie strednej skrutky M5//
        380:
            SC_P1_Srobovanie.StepName:='380 - Automaticky Rezim - model 5H, napolohovanie strednej skrutkovacky M5 na poziciu odobratia sroby M5 zo zasobnika';
            SC_P1_Srobovanie.IdleTime.PT:= T#200ms;
            SC_P1_Srobovanie.AlarmTime.PT:= T#5s;

            P1_Robot.KOM_OUT.ManipSrobovania_BezpecnaPozicia:= FALSE;

            P1_Srobovanie.PAR.OsX_ZadanaPozicia:= P1_RemPremenne.P1_Srob5H_PozX_OdobratSkrutkyM5; //mm
            P1_Srobovanie.PAR.OsY_ZadanaPozicia:= P1_RemPremenne.P1_Srob5H_PozY_OdobratSkrutkyM5; //mm

            IF NOT SC_P1_Srobovanie.Switch1 AND SC_OvlManipulatora_OsX.Step = 1 AND P1_Srobovacky_VychodziaPozicia AND Safety.STAV.P1_ZonaBunky_AKTIVNA THEN
                OsX_POLOHUJ:= TRUE;
                SC_P1_Srobovanie.Switch1:= TRUE;
            END_IF

            IF NOT SC_P1_Srobovanie.Switch2 AND SC_OvlManipulatora_OsY.Step = 1 AND P1_Srobovacky_VychodziaPozicia AND (P1_Srobovanie.ServoManipulOsX_M20.STATUS.ActualPosition > 14) AND Safety.STAV.P1_ZonaBunky_AKTIVNA THEN
                OsY_POLOHUJ:= TRUE;
                SC_P1_Srobovanie.Switch2:= TRUE;
            END_IF

            IF P1_Srobovanie.STAV.OsX_PoziciaDosiahnuta AND P1_Srobovanie.STAV.OsY_PoziciaDosiahnuta THEN
                P1_Srobovanie.STAV.OsX_PoziciaDosiahnuta:= FALSE;
                P1_Srobovanie.STAV.OsY_PoziciaDosiahnuta:= FALSE;
                SC_P1_Srobovanie.ResetStep:= TRUE;
                SC_P1_Srobovanie.Step:= 382;
            END_IF

        382:
            SC_P1_Srobovanie.StepName:='382 - Automaticky Rezim - model 5H, kontrola skrutky M5 na vystupe podavaca';
            SC_P1_Srobovanie.IdleTime.PT:= T#200ms;
            SC_P1_Srobovanie.AlarmTime.PT:= T#10s;
            SC_P1_Srobovanie.AlarmTime.IN:= TRUE;

            IF P1_Srobovanie.SkrutkovaciSet_M5.SkrutkaM5_Pripravena AND P1_Srobovanie.IN.OddelSrobM5_SrobaNaVystupe_OS14 THEN
                SC_P1_Srobovanie.ResetStep:= TRUE;
                SC_P1_Srobovanie.Step:= 383;
            ELSIF SC_P1_Srobovanie.AlarmTime.Q THEN
                P1_Alarmy[120]:= TRUE;
                P1_StoperSrobovania.STAV.Porucha:= TRUE;
                P1_Srobovanie.OUT.KOM_Srobovanie_Ukoncene:= TRUE;
                SC_P1_Srobovanie.ResetStep:= TRUE;
                SC_P1_Srobovanie.Step:= 393;
            END_IF

        383:
            SC_P1_Srobovanie.StepName:='383 - Automaticky Rezim - model 5H, odobratie skrutky M5 z podavaca';
            SC_P1_Srobovanie.IdleTime.PT:= T#200ms;
            SC_P1_Srobovanie.AlarmTime.PT:= T#5s;

            SC_P1_Srobovanie.IdleTime.IN:= P1_Srobovanie.IN.SkrutkM5_SnimacVakua_S28;

            IF NOT SC_P1_Srobovanie.Switch1 THEN
                P1_Srobovanie.OUT.SkrutkM5_VYSUN_YV104:= TRUE;
                P1_Srobovanie.OUT.SkrutkM5_PrisavSkrut_VYPNI_YV109:= FALSE;
                P1_Srobovanie.OUT.SkrutkM5_PrisavSkrut_ZAPNI_YV105:= TRUE;
                SC_P1_Srobovanie.IdleTime.IN:= TRUE;
                SC_P1_Srobovanie.Switch1:= TRUE;
            END_IF

            IF SC_P1_Srobovanie.IdleTime.Q THEN
                SC_P1_Srobovanie.ResetStep:= TRUE;
                SC_P1_Srobovanie.Step:= 384;
            END_IF

        384:
            SC_P1_Srobovanie.StepName:='384 - Automaticky Rezim - model 5H, zasunutie skrutkovacky M5, vystavenie signalu skrutka odobrata';
            SC_P1_Srobovanie.IdleTime.PT:= T#200ms;
            SC_P1_Srobovanie.AlarmTime.PT:= T#5s;

            IF NOT SC_P1_Srobovanie.Switch1 THEN
                P1_Srobovanie.OUT.SkrutkM5_VYSUN_YV104:= FALSE;
                SC_P1_Srobovanie.Switch1:= TRUE;
            END_IF

            IF P1_Srobovanie.IN.SkrutkM5_ZASUNUTY_MS39 THEN
                P1_Srobovanie.SkrutkovaciSet_M5.SkrutkaM5_Odobrata:= TRUE;
                SC_P1_Srobovanie.ResetStep:= TRUE;
                SC_P1_Srobovanie.Step:= 385;
            END_IF

        385:
            SC_P1_Srobovanie.StepName:='385 - Automaticky Rezim - model 5H, cakam na zrusenie signalu skrutka M5 pripravena';
            SC_P1_Srobovanie.IdleTime.PT:= T#200ms;
            SC_P1_Srobovanie.AlarmTime.PT:= T#5s;

            IF NOT P1_Srobovanie.SkrutkovaciSet_M5.SkrutkaM5_Pripravena THEN
                P1_Srobovanie.SkrutkovaciSet_M5.SkrutkaM5_Odobrata:= FALSE;
                SC_P1_Srobovanie.ResetStep:= TRUE;
                SC_P1_Srobovanie.Step:= 386;
            END_IF

        386:
            SC_P1_Srobovanie.StepName:='386 - Automaticky Rezim - model 5H, napolohovanie strednej skrutkovacky M5 na poziciu strednej skrutky M5';
            SC_P1_Srobovanie.IdleTime.PT:= T#200ms;
            SC_P1_Srobovanie.AlarmTime.PT:= T#5s;

            P1_Robot.KOM_OUT.ManipSrobovania_BezpecnaPozicia:= FALSE;

            P1_Srobovanie.PAR.OsX_ZadanaPozicia:= P1_RemPremenne.P1_Srob5H_PozX_StrednejSkrutkyM5; //mm
            P1_Srobovanie.PAR.OsY_ZadanaPozicia:= P1_RemPremenne.P1_Srob5H_PozY_StrednejSkrutkyM5; //mm

            IF NOT SC_P1_Srobovanie.Switch1 AND SC_OvlManipulatora_OsX.Step = 1 AND P1_Srobovacky_VychodziaPozicia AND Safety.STAV.P1_ZonaBunky_AKTIVNA THEN
                OsX_POLOHUJ:= TRUE;
                SC_P1_Srobovanie.Switch1:= TRUE;
            END_IF

            IF NOT SC_P1_Srobovanie.Switch2 AND SC_OvlManipulatora_OsY.Step = 1 AND P1_Srobovacky_VychodziaPozicia AND (P1_Srobovanie.ServoManipulOsX_M20.STATUS.ActualPosition > 14) AND Safety.STAV.P1_ZonaBunky_AKTIVNA THEN
                OsY_POLOHUJ:= TRUE;
                SC_P1_Srobovanie.Switch2:= TRUE;
            END_IF

            IF P1_Srobovanie.STAV.OsX_PoziciaDosiahnuta AND P1_Srobovanie.STAV.OsY_PoziciaDosiahnuta THEN
                P1_Srobovanie.STAV.OsX_PoziciaDosiahnuta:= FALSE;
                P1_Srobovanie.STAV.OsY_PoziciaDosiahnuta:= FALSE;
                IF P1_Srobovanie.RR_PolohujNaPoziciuSkrutky_5H THEN
                    P1_Srobovanie.RR_PolohujNaPoziciuSkrutky_5H:= FALSE;
                    P1_Srobovanie.RR_PolohujNaPoziciuSkrutky_4F:= FALSE;
                    P1_Srobovanie.RR_PolohujNaPoziciuSkrutky_5F:= FALSE;
                    SC_P1_Srobovanie.ResetStep:= TRUE;
                    SC_P1_Srobovanie.Step:= 700;
                ELSE
                    SC_P1_Srobovanie.ResetStep:= TRUE;
                    SC_P1_Srobovanie.Step:= 387;
                END_IF
            END_IF

        387:
            SC_P1_Srobovanie.StepName:='387 - Automaticky Rezim - model 5H, vymazanie vysledkov srobovania';
            SC_P1_Srobovanie.IdleTime.PT:= T#2s;
            SC_P1_Srobovanie.AlarmTime.PT:= T#5s;

            IF NOT SC_P1_Srobovanie.Switch1 THEN
                P1_Srobovanie.Skrutkovacka_M5.RESET_Vysledkov:= TRUE;
                SC_P1_Srobovanie.Switch1:= TRUE;
            END_IF

            IF NOT P1_Srobovanie.Skrutkovacka_M5.Stav_VysledokUtahovania_NG AND NOT P1_Srobovanie.Skrutkovacka_M5.Stav_VysledokUtahovania_OK  THEN
                P1_Srobovanie.Skrutkovacka_M5.RESET_Vysledkov:= FALSE;
                SC_P1_Srobovanie.ResetStep:= TRUE;
                SC_P1_Srobovanie.Step:= 388;
            END_IF

        388:
            SC_P1_Srobovanie.StepName:='388 - Automaticky Rezim - model 5H, prepnutie programu';
            SC_P1_Srobovanie.IdleTime.PT:= T#2s;
            SC_P1_Srobovanie.AlarmTime.PT:= T#10s;

            IF NOT SC_P1_Srobovanie.Switch1 THEN
                P1_Srobovanie.Skrutkovacka_M5.CisloZadanehoProgramu:= 1;
                SC_P1_Srobovanie.AlarmTime.IN:= TRUE;
                SC_P1_Srobovanie.Switch1:= TRUE;
            END_IF

            IF P1_Srobovanie.Skrutkovacka_M5.Stav_CisloAktualnehoProgramu = 1 AND P1_Srobovanie.Skrutkovacka_M5.Stav_READY_to_START AND NOT P1_Srobovanie.Skrutkovacka_M5.Stav_UtahovanieUkoncene THEN
                SC_P1_Srobovanie.ResetStep:= TRUE;
                SC_P1_Srobovanie.Step:= 389;
            ELSIF SC_P1_Srobovanie.AlarmTime.Q AND NOT P1_Srobovanie.Skrutkovacka_M5.Stav_READY_to_START THEN
                P1_Alarmy[150]:= TRUE;
                P1_StoperSrobovania.STAV.Porucha:= TRUE;
                P1_Srobovanie.OUT.KOM_Srobovanie_Ukoncene:= TRUE;
                SC_P1_Srobovanie.ResetStep:= TRUE;
                SC_P1_Srobovanie.Step:= 393;
            END_IF

        389:
            SC_P1_Srobovanie.StepName:='389 - Automaticky Rezim - model 5H, vysunutie skrutkovacky M5';
            SC_P1_Srobovanie.IdleTime.PT:= T#2s;
            SC_P1_Srobovanie.AlarmTime.PT:= T#5s;

            SC_P1_Srobovanie.AlarmTime.IN:= (P1_Srobovanie.IN.SkrutkM5_VysunutieHrotu_IOS9 < 2);

            IF NOT SC_P1_Srobovanie.Switch1 THEN
                P1_Srobovanie.OUT.SkrutkM5_VYSUN_YV104:= TRUE;
                P1_Srobovanie.Skrutkovacka_M5.START_Utahovania:= TRUE;
                SC_P1_Srobovanie.Switch1:= TRUE;
            END_IF

            IF NOT P1_Srobovanie.Skrutkovacka_M5.Stav_UtahovanieUkoncene AND P1_Srobovanie.IN.SkrutkM5_VysunutieHrotu_IOS9 > 2 AND NOT TEST THEN
                SC_P1_Srobovanie.ResetStep:= TRUE;
                SC_P1_Srobovanie.Step:= 390;
            ELSIF SC_P1_Srobovanie.AlarmTime.Q AND NOT TEST THEN
                P1_Alarmy[143]:= TRUE;
                P1_Srobovanie.OUT.SkrutkM5_VYSUN_YV104:= FALSE;
                P1_Srobovanie.Skrutkovacka_M5.START_Utahovania:= FALSE;
                P1_StoperSrobovania.STAV.Porucha:= TRUE;
                P1_Srobovanie.OUT.KOM_Srobovanie_Ukoncene:= TRUE;
                SC_P1_Srobovanie.ResetStep:= TRUE;
                SC_P1_Srobovanie.Step:= 393;
            END_IF

        390:
            SC_P1_Srobovanie.StepName:='390 - Automaticky Rezim - model 5H, cakam na ukoncenie skrutkovania skrutkovacky M5';
            SC_P1_Srobovanie.IdleTime.PT:= T#30s;
            SC_P1_Srobovanie.AlarmTime.PT:= T#10s;
            SC_P1_Srobovanie.IdleTime.IN:= TRUE;
            SC_P1_Srobovanie.AlarmTime.IN:= TRUE;

            IF P1_Srobovanie.Skrutkovacka_M5.Stav_UtahovanieUkoncene THEN
                P1_Srobovanie.Skrutkovacka_M5.START_Utahovania:= FALSE;
                CasSrobovania:= TIME_TO_REAL(SC_P1_Srobovanie.IdleTime.ET);
                Reports.Skrutkovacky.VyskaSkrutkovania.P1_StrednaSkrutkaM5:= REAL_TO_STRING(P1_Srobovanie.IN.SkrutkM5_VysunutieHrotu_IOS9);
                Reports.Skrutkovacky.CasSkrutkovania.P1_StrednaSkrutkaM5:= REAL_TO_STRING(CasSrobovania/1000);
                SC_P1_Srobovanie.ResetStep:= TRUE;
                SC_P1_Srobovanie.Step:= 391;
            ELSIF SC_P1_Srobovanie.AlarmTime.Q THEN
                P1_Alarmy[147]:= TRUE;
                P1_Srobovanie.OUT.SkrutkM5_VYSUN_YV104:= FALSE;
                P1_Srobovanie.Skrutkovacka_M5.START_Utahovania:= FALSE;
                P1_StoperSrobovania.STAV.Porucha:= TRUE;
                P1_Srobovanie.OUT.KOM_Srobovanie_Ukoncene:= TRUE;
                SC_P1_Srobovanie.ResetStep:= TRUE;
                SC_P1_Srobovanie.Step:= 393;
            END_IF

        391:
            SC_P1_Srobovanie.StepName:='391 - Automaticky Rezim - model 5H, zasunutie skrutkovacky M5 a vypnutie prisavania skrutky';
            SC_P1_Srobovanie.IdleTime.PT:= T#200ms;
            SC_P1_Srobovanie.AlarmTime.PT:= T#5s;

            IF NOT SC_P1_Srobovanie.Switch1 THEN
                P1_Srobovanie.OUT.SkrutkM5_VYSUN_YV104:= FALSE;
                P1_Srobovanie.OUT.SkrutkM5_PrisavSkrut_ZAPNI_YV105:= FALSE;
                P1_Srobovanie.OUT.SkrutkM5_PrisavSkrut_VYPNI_YV109:= TRUE;
                SC_P1_Srobovanie.Switch1:= TRUE;
            END_IF

            IF P1_Srobovanie.IN.SkrutkM5_ZASUNUTY_MS39 THEN
                SC_P1_Srobovanie.ResetStep:= TRUE;
                SC_P1_Srobovanie.Step:= 392;
            END_IF

        392:
            SC_P1_Srobovanie.StepName:='392 - Automaticky Rezim - model 5H, kontrola vysledkov skrutkovania pravej skrutky M5';
            SC_P1_Srobovanie.IdleTime.PT:= T#200ms;
            SC_P1_Srobovanie.AlarmTime.PT:= T#5s;

            IF P1_Srobovanie.Skrutkovacka_M5.Stav_VysledokUtahovania_OK THEN
                P1_Srobovanie.STAV.Vysledok_Srobovania:= 'OK';
                P1_Srobovanie.OUT.KOM_Srobovanie_Ukoncene:= TRUE;
                SC_P1_Srobovanie.ResetStep:= TRUE;
                SC_P1_Srobovanie.Step:= 393;
            ELSIF P1_Srobovanie.Skrutkovacka_M5.Stav_VysledokUtahovania_NG THEN
                P1_Srobovanie.STAV.Vysledok_Srobovania:= 'NG';
                P1_Srobovanie.OUT.KOM_Srobovanie_Ukoncene:= TRUE;
                SC_P1_Srobovanie.ResetStep:= TRUE;
                SC_P1_Srobovanie.Step:= 393;
            END_IF

        393:
            SC_P1_Srobovanie.StepName:='393 - Automaticky Rezim - model 5H, cakam na zrusenie signalu zaskrutkuj strednu skrutku M5';
            SC_P1_Srobovanie.IdleTime.PT:= T#200ms;
            SC_P1_Srobovanie.AlarmTime.PT:= T#5s;

            IF NOT P1_StoperSrobovania.OUT.KOM_5H_ZasrobujStrednuSkrutku_M5 THEN
                P1_Srobovanie.OUT.KOM_Srobovanie_Ukoncene:= FALSE;
                SC_P1_Srobovanie.ResetStep:= TRUE;
                SC_P1_Srobovanie.Step:= 100;
            END_IF

            //Presun manipulátora do pozície VPRED//

        400:
            SC_P1_Srobovanie.StepName:='400 - Automaticky Rezim - napolohovanie manipulatora do prednej pozicie';
            SC_P1_Srobovanie.IdleTime.PT:= T#200ms;
            SC_P1_Srobovanie.AlarmTime.PT:= T#5s;

            P1_Robot.KOM_OUT.ManipSrobovania_BezpecnaPozicia:= FALSE;

            P1_Srobovanie.PAR.OsX_ZadanaPozicia:= 15; //mm
            P1_Srobovanie.PAR.OsY_ZadanaPozicia:= 310; //mm

            IF NOT SC_P1_Srobovanie.Switch1 AND SC_OvlManipulatora_OsX.Step = 1 AND P1_Srobovacky_VychodziaPozicia AND Safety.STAV.P1_ZonaBunky_AKTIVNA THEN
                OsX_POLOHUJ:= TRUE;
                SC_P1_Srobovanie.Switch1:= TRUE;
            END_IF

            IF NOT SC_P1_Srobovanie.Switch2 AND SC_OvlManipulatora_OsY.Step = 1 AND P1_Srobovacky_VychodziaPozicia AND (P1_Srobovanie.ServoManipulOsX_M20.STATUS.ActualPosition > 14) AND Safety.STAV.P1_ZonaBunky_AKTIVNA THEN
                OsY_POLOHUJ:= TRUE;
                SC_P1_Srobovanie.Switch2:= TRUE;
            END_IF

            IF P1_Srobovanie.STAV.OsX_PoziciaDosiahnuta AND P1_Srobovanie.STAV.OsY_PoziciaDosiahnuta THEN
                P1_Srobovanie.STAV.OsX_PoziciaDosiahnuta:= FALSE;
                P1_Srobovanie.STAV.OsY_PoziciaDosiahnuta:= FALSE;
                P1_Srobovanie.OUT.KOM_PresunVPRED_Ukonceny:= TRUE;
                SC_P1_Srobovanie.ResetStep:= TRUE;
                SC_P1_Srobovanie.Step:= 402;
            END_IF

        402:
            SC_P1_Srobovanie.StepName:='402 - Automaticky Rezim - cakam na zrusenie signalu presun manipulatora do prednej pozicie';
            SC_P1_Srobovanie.IdleTime.PT:= T#200ms;
            SC_P1_Srobovanie.AlarmTime.PT:= T#5s;

            IF NOT P1_StoperSrobovania.OUT.KOM_PresunManipulator_DOPREDU THEN
                SC_P1_Srobovanie.ResetStep:= TRUE;
                SC_P1_Srobovanie.Step:= 100;
            END_IF

            //Presun manipulatora do pozicie VZAD//

        420:
            SC_P1_Srobovanie.StepName:='420 - Automaticky Rezim - napolohovanie manipulatora do zadnej pozicie';
            SC_P1_Srobovanie.IdleTime.PT:= T#200ms;
            SC_P1_Srobovanie.AlarmTime.PT:= T#5s;

            P1_Robot.KOM_OUT.ManipSrobovania_BezpecnaPozicia:= FALSE;

            P1_Srobovanie.PAR.OsX_ZadanaPozicia:= 15; //mm
            P1_Srobovanie.PAR.OsY_ZadanaPozicia:= 0; //mm

            IF NOT SC_P1_Srobovanie.Switch1 AND SC_OvlManipulatora_OsX.Step = 1 AND P1_Srobovacky_VychodziaPozicia AND Safety.STAV.P1_ZonaBunky_AKTIVNA THEN
                OsX_POLOHUJ:= TRUE;
                SC_P1_Srobovanie.Switch1:= TRUE;
            END_IF

            IF NOT SC_P1_Srobovanie.Switch2 AND SC_OvlManipulatora_OsY.Step = 1 AND P1_Srobovacky_VychodziaPozicia AND (P1_Srobovanie.ServoManipulOsX_M20.STATUS.ActualPosition > 14) AND Safety.STAV.P1_ZonaBunky_AKTIVNA THEN
                OsY_POLOHUJ:= TRUE;
                SC_P1_Srobovanie.Switch2:= TRUE;
            END_IF

            IF P1_Srobovanie.STAV.OsX_PoziciaDosiahnuta AND P1_Srobovanie.STAV.OsY_PoziciaDosiahnuta THEN
                P1_Srobovanie.STAV.OsX_PoziciaDosiahnuta:= FALSE;
                P1_Srobovanie.STAV.OsY_PoziciaDosiahnuta:= FALSE;
                P1_Srobovanie.OUT.KOM_PresunVZAD_Ukonceny:= TRUE;
                SC_P1_Srobovanie.ResetStep:= TRUE;
                SC_P1_Srobovanie.Step:= 422;
            END_IF

        422:
            SC_P1_Srobovanie.StepName:='422 - Automaticky Rezim - cakam na zrusenie signalu presun manipulatora do zadnej pozicie';
            SC_P1_Srobovanie.IdleTime.PT:= T#200ms;
            SC_P1_Srobovanie.AlarmTime.PT:= T#5s;

            IF NOT P1_StoperSrobovania.OUT.KOM_PresunManipulator_DOZADU THEN
                SC_P1_Srobovanie.ResetStep:= TRUE;
                SC_P1_Srobovanie.Step:= 100;
            END_IF

            //*********************************************************Čistenie skrutkovačiek*****************************************************************************//

            //Čistenie skrutkovačky K30//
        500:
            SC_P1_Srobovanie.StepName:='500 - Automaticky Rezim - cistenie skrutkovacky K30';
            SC_P1_Srobovanie.IdleTime.PT:= T#200ms;
            SC_P1_Srobovanie.AlarmTime.PT:= T#5s;

            P1_Srobovanie.PAR.OsX_ZadanaPozicia:= 15; //mm
            P1_Srobovanie.PAR.OsY_ZadanaPozicia:= 0; //mm

            IF NOT SC_P1_Srobovanie.Switch1 AND SC_OvlManipulatora_OsX.Step = 1 AND P1_Srobovacky_VychodziaPozicia AND Safety.STAV.P1_ZonaBunky_AKTIVNA THEN
                P1_Srobovanie.SkrutkovaciSet_K30.SkrutkaK30_Odobrata:= FALSE;
                P1_Srobovanie.SkrutkovaciSet_K30.Automat:= TRUE;
                P1_Srobovanie.SkrutkovaciSet_K30.Reset:= TRUE;
                OsX_POLOHUJ:= TRUE;
                SC_P1_Srobovanie.Switch1:= TRUE;
            END_IF
```
